// TIA Portal project "Semafoare_2026" (V15.1)

(* hardware
DEVICE "S71500/ET200MP station_1"  S7-1500 station
   slot 0: "Rail_0"  Rack  6ES7 590-1***0-0AA0
   slot 1: "PLC_1"  CPU 1513-1 PN  6ES7 513-1AL02-0AB0  V2.6
      slot 3: "CPU display_1"  6ES7591-1AA00-0AA0
DEVICE "HMI_1"  KTP900 Basic PN
   slot 0: "HMI_1"  KTP900 Basic PN  6AV2 123-2JB03-0AX0  15.1.0.0
   slot 1: "HMI_RT_1"  KTP900 Basic PN  6AV2 123-2JB03-0AX0  15.1.0.0
   slot 5: "HMI_1.IE_CP_1"  PROFINET Interface  15.0.1.0
      slot 1: "PROFINET Interface_1"  PROFINET Interface
         slot 1: "Port_1"  Port
*)

// ===== PLC "PLC_1"  CPU 1513-1 PN =====

VAR_GLOBAL   // PLC tag table "Default tag table"
   "Clock_Byte" AT %MB0 : Byte;
   "Clock_10Hz" AT %M0.0 : Bool;
   "Clock_5Hz" AT %M0.1 : Bool;
   "Clock_2.5Hz" AT %M0.2 : Bool;
   "Clock_2Hz" AT %M0.3 : Bool;
   "Clock_1.25Hz" AT %M0.4 : Bool;
   "Clock_1Hz" AT %M0.5 : Bool;
   "Clock_0.625Hz" AT %M0.6 : Bool;
   "Clock_0.5Hz" AT %M0.7 : Bool;
END_VAR

DATA_BLOCK "Semafor_masini_ciclu_DB"   // DB1
{ S7_Optimized_Access := 'TRUE' }
VERSION : 0.1
   VAR
      rosu_on : Bool;
      galben_on : Bool;
      galben_on_hmi : Bool;
      verde_on : Bool;
      time_elapsed_rosu : Time;
      time_elapsed_rosu_secunde : Time;
      time_elapsed_verde : Time;
      time_elapsed_verde_secunde : Time;
      time_elapsed_galben : Time;
      time_elapsed_galben_secunde : Time;
      "mod" : Int;
   END_VAR
BEGIN
END_DATA_BLOCK

DATA_BLOCK "Semafor_pietoni_DB"   // DB2
{ S7_Optimized_Access := 'TRUE' }
VERSION : 0.1
   VAR
      "mod" : Int;
      rosu_on : Bool;
      verde_on : Bool;
      time_elapsed_rosu : Time;
      time_elapsed_sec_rosu : Time;
      time_elapsed_verde : Time;
      time_elapsed_sec_verde : Time;
   END_VAR
BEGIN
END_DATA_BLOCK

DATA_BLOCK "Semafor_masini_ciclu_DB_1"   // DB3
{ S7_Optimized_Access := 'TRUE' }
VERSION : 0.1
// stored: InstanceOfName Semafor_masini_ciclu
"Semafor_masini_ciclu"
BEGIN
END_DATA_BLOCK

DATA_BLOCK "Semafor_pietoni_DB_1"   // DB4
{ S7_Optimized_Access := 'TRUE' }
VERSION : 0.1
// stored: InstanceOfName Semafor_pietoni
"Semafor_pietoni"
BEGIN
END_DATA_BLOCK

DATA_BLOCK "Semafor_pietoni_buton_DB"   // DB5
{ S7_Optimized_Access := 'TRUE' }
VERSION : 0.1
   VAR
      "mod" : Int;
      rosu_on : Bool;
      verde_on : Bool;
      buton : Bool;
      timer_buton_gata : Bool;
      intermitent_hmi : Bool;
      vizibil_hmi : Bool;
      time_elapsed_verde : Time;
      time_elapsed_sec_verde : Time;
      timp_intre : Time;
      timp_intre_sec : Time;
   END_VAR
BEGIN
END_DATA_BLOCK

DATA_BLOCK "Semafor_pietoni_buton_DB_1"   // DB6
{ S7_Optimized_Access := 'TRUE' }
VERSION : 0.1
// stored: InstanceOfName Semafor_pietoni_buton
"Semafor_pietoni_buton"
BEGIN
END_DATA_BLOCK

DATA_BLOCK "Semafor_masina_pietoni_DB"   // DB7
{ S7_Optimized_Access := 'TRUE' }
VERSION : 0.1
   VAR
      "mod" : Int;
      timer_buton_gata : Bool;
      buton : Bool;
      verde_on : Bool;
      rosu_on : Bool;
      galben_on : Bool;
      galben_on_hmi : Bool;
      pieton_verde_on : Bool;
      pieton_rosu_on : Bool;
      intermitent_hmi : Bool;
      vizibil_hmi : Bool;
      time_elapsed_galben : Time;
      time_elapsed_galben_sec : Time;
      time_elapsed_rosu : Time;
      time_elapsed_rosu_sec : Time;
      pieton_time_elapsed_verde : Time;
      pieton_time_elapsed_verde_sec : Time;
      time_intre : Time;
      time_buton : Time;
   END_VAR
BEGIN
END_DATA_BLOCK

DATA_BLOCK "Semafor_masina_buton_DB"   // DB8
{ S7_Optimized_Access := 'TRUE' }
VERSION : 0.1
   VAR
      verde_on : Bool;
      rosu_on : Bool;
      galben_on : Bool;
      galben_on_hmi : Bool;
      time_elapsed_galben : Time;
      time_elapsed_rosu : Time;
      time_elapsed_galben_sec : Time;
      tine_elapsed_rosu_sec : Time;
   END_VAR
BEGIN
END_DATA_BLOCK

DATA_BLOCK "Semafor_masina_buton_DB_1"   // DB9
{ S7_Optimized_Access := 'TRUE' }
VERSION : 0.1
// stored: InstanceOfName Semafor_masina_buton
"Semafor_masina_buton"
BEGIN
END_DATA_BLOCK

DATA_BLOCK "Semafor_masina_pietoni_DB_1"   // DB10
{ S7_Optimized_Access := 'TRUE' }
VERSION : 0.1
// stored: InstanceOfName Semafor_masina_pietoni
"Semafor_masina_pietoni"
BEGIN
END_DATA_BLOCK

DATA_BLOCK "Semafor_masina_buton_DB_2"   // DB11
{ S7_Optimized_Access := 'TRUE' }
VERSION : 0.1
// stored: InstanceOfName Semafor_masina_buton
"Semafor_masina_buton"
BEGIN
END_DATA_BLOCK

DATA_BLOCK "Semafor_pietoni_buton_DB_2"   // DB12
{ S7_Optimized_Access := 'TRUE' }
VERSION : 0.1
// stored: InstanceOfName Semafor_pietoni_buton
"Semafor_pietoni_buton"
BEGIN
END_DATA_BLOCK

DATA_BLOCK "Clock_custom_0.7Hz_DB"   // DB13
{ S7_Optimized_Access := 'TRUE' }
VERSION : 0.1
// stored: InstanceOfName Clock_custom_0.7Hz
"Clock_custom_0.7Hz"
BEGIN
END_DATA_BLOCK

DATA_BLOCK "test"   // DB14
{ S7_Optimized_Access := 'TRUE' }
VERSION : 0.1
   VAR
      activ : Bool;
      re : Bool;
      "counter" : Int;
   END_VAR
BEGIN
END_DATA_BLOCK

DATA_BLOCK "Buzzer_DB"   // DB15
{ S7_Optimized_Access := 'TRUE' }
VERSION : 0.1
   VAR
      permisiune_plecare : Bool;
      pornire_sunet : Bool;
   END_VAR
BEGIN
END_DATA_BLOCK

DATA_BLOCK "Buzzer_DB_1"   // DB16
{ S7_Optimized_Access := 'TRUE' }
VERSION : 0.1
// stored: InstanceOfName Buzzer
"Buzzer"
BEGIN
END_DATA_BLOCK

DATA_BLOCK "Buzzer_Pieton_buton_DB"   // DB17
{ S7_Optimized_Access := 'TRUE' }
VERSION : 0.1
   VAR
      permisiune_plecare : Bool;
      pornire_sunet : Bool;
   END_VAR
BEGIN
END_DATA_BLOCK

DATA_BLOCK "Buzzer_pieton_Masina_buton_DB"   // DB18
{ S7_Optimized_Access := 'TRUE' }
VERSION : 0.1
   VAR
      permisiune_plecare : Bool;
      pornire_sunet : Bool;
   END_VAR
BEGIN
END_DATA_BLOCK

DATA_BLOCK "Buzzer_DB_2"   // DB19
{ S7_Optimized_Access := 'TRUE' }
VERSION : 0.1
// stored: InstanceOfName Buzzer
"Buzzer"
BEGIN
END_DATA_BLOCK

DATA_BLOCK "Buzzer_DB_3"   // DB20
{ S7_Optimized_Access := 'TRUE' }
VERSION : 0.1
// stored: InstanceOfName Buzzer
"Buzzer"
BEGIN
END_DATA_BLOCK

DATA_BLOCK "Semafoare-2-masini_DB"   // DB21
{ S7_Optimized_Access := 'TRUE' }
VERSION : 0.1
   VAR
      "mod" : Int;
      te_rosu_1 : Time;
      te_rosu_sec_1 : Time;
      te_rosu_2 : Time;
      te_rosu_sec_2 : Time;
      te_galben_1 : Time;
      te_galben_sec_1 : Time;
      te_galben_2 : Time;
      te_galben_sec_2 : Time;
      te_verde_1 : Time;
      te_verde_sec_1 : Time;
      te_verde_2 : Time;
      te_verde_sec_2 : Time;
      verde_on_1 : Bool;
      verde_on_2 : Bool;
      galben_on_1 : Bool;
      galben_hmi_on_1 : Bool;
      galben_on_2 : Bool;
      galben_hmi_on_2 : Bool;
      rosu_on_1 : Bool;
      rosu_on_2 : Bool;
   END_VAR
BEGIN
END_DATA_BLOCK

DATA_BLOCK "Semafoare-2-masini_DB_1"   // DB22
{ S7_Optimized_Access := 'TRUE' }
VERSION : 0.1
// stored: InstanceOfName Semafoare-2-masini
"Semafoare-2-masini"
BEGIN
END_DATA_BLOCK

DATA_BLOCK "Semafor_masini_ciclu_DB_2"   // DB23
{ S7_Optimized_Access := 'TRUE' }
VERSION : 0.1
// stored: InstanceOfName Semafor_masini_ciclu
"Semafor_masini_ciclu"
BEGIN
END_DATA_BLOCK

DATA_BLOCK "Semafor_masini_ciclu_DB_3"   // DB24
{ S7_Optimized_Access := 'TRUE' }
VERSION : 0.1
// stored: InstanceOfName Semafor_masini_ciclu
"Semafor_masini_ciclu"
BEGIN
END_DATA_BLOCK

DATA_BLOCK "Semafor_masini_1_DB"   // DB25
{ S7_Optimized_Access := 'TRUE' }
VERSION : 0.1
// stored: InstanceOfName Semafor_masini_1
"Semafor_masini_1"
BEGIN
END_DATA_BLOCK

DATA_BLOCK "Semafor_masina_2_DB"   // DB26
{ S7_Optimized_Access := 'TRUE' }
VERSION : 0.1
// stored: InstanceOfName Semafor_masina_2
"Semafor_masina_2"
BEGIN
END_DATA_BLOCK

FUNCTION_BLOCK "Semafor_masini_ciclu"   // FB1, LAD
{ S7_Optimized_Access := 'TRUE' }
VERSION : 0.1
   VAR_INPUT
      mod_functinare : Int;
   END_VAR
   VAR_OUTPUT
      time_elapsed_verde : Time;
      time_elapsed_galben : Time;
      time_elapsed_rosu : Time;
   END_VAR
   VAR_IN_OUT
      verde_on : Bool;
      rosu_on : Bool;
      galben_on : Bool;
   END_VAR
   VAR
      timer_rosu : TON_TIME;
      timer_galben : TON_TIME;
      timer_verde : TON_TIME;
      galben_intermitent_on : Bool;
      re1 : Bool;
      re_aux : Bool;
      mod_normal : Bool;
      reseteaza_ciclul : Bool;
      porneste_verde : Bool;
      porneste_rosu : Bool;
      porneste_galben : Bool;
   END_VAR
   VAR_TEMP   // added for the SCL form of the ladder/FBD networks
      _w1 : Bool;
   END_VAR
BEGIN

REGION Network 1: semafor modul normal/mod oprire
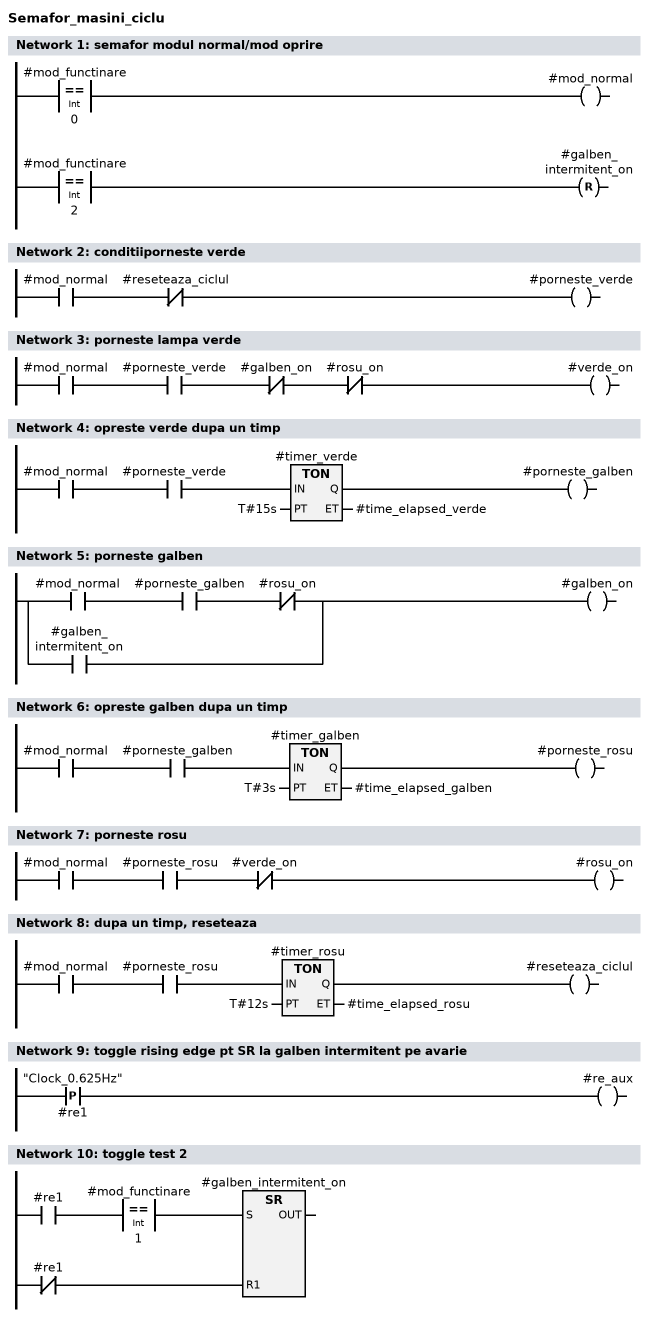
   RUNG wire#powerrail
      { S7_Templates := "SrcType := Int" } EQ_Contact(in1 := #mod_functinare, in2 := 0)
      Coil( #mod_normal )
   END_RUNG
   RUNG wire#powerrail
      { S7_Templates := "SrcType := Int" } EQ_Contact(in1 := #mod_functinare, in2 := 2)
      R_Coil( #galben_intermitent_on )
   END_RUNG
   // the same network as SCL:
   #mod_normal := #mod_functinare = 0;
   IF #mod_functinare = 2 THEN #galben_intermitent_on := FALSE; END_IF;
END_REGION

REGION Network 2: conditiiporneste verde
   RUNG wire#powerrail
      Contact( #mod_normal )
      I_Contact( #reseteaza_ciclul )
      Coil( #porneste_verde )
   END_RUNG
   // the same network as SCL:
   #porneste_verde := #mod_normal AND NOT #reseteaza_ciclul;
END_REGION

REGION Network 3: porneste lampa verde
   RUNG wire#powerrail
      Contact( #mod_normal )
      Contact( #porneste_verde )
      I_Contact( #galben_on )
      I_Contact( #rosu_on )
      Coil( #verde_on )
   END_RUNG
   // the same network as SCL:
   #verde_on := #mod_normal AND #porneste_verde AND NOT #galben_on AND NOT #rosu_on;
END_REGION

REGION Network 4: opreste verde dupa un timp
   #timer_verde(IN := #mod_normal AND #porneste_verde, PT := T#15s, ET => #time_elapsed_verde);   // TON
   #porneste_galben := #timer_verde.Q;
END_REGION

REGION Network 5: porneste galben
   RUNG wire#powerrail
      Contact( #mod_normal )
      Contact( #porneste_galben )
      I_Contact( #rosu_on )
      wire#w1
      Coil( #galben_on )
   END_RUNG
   RUNG wire#powerrail
      Contact( #galben_intermitent_on )
   END_RUNG wire#w1
   // the same network as SCL:
   #galben_on := (#mod_normal AND #porneste_galben AND NOT #rosu_on) OR #galben_intermitent_on;
END_REGION

REGION Network 6: opreste galben dupa un timp
   #timer_galben(IN := #mod_normal AND #porneste_galben, PT := T#3s, ET => #time_elapsed_galben);   // TON
   #porneste_rosu := #timer_galben.Q;
END_REGION

REGION Network 7: porneste rosu
   RUNG wire#powerrail
      Contact( #mod_normal )
      Contact( #porneste_rosu )
      I_Contact( #verde_on )
      Coil( #rosu_on )
   END_RUNG
   // the same network as SCL:
   #rosu_on := #mod_normal AND #porneste_rosu AND NOT #verde_on;
END_REGION

REGION Network 8: dupa un timp, reseteaza
   #timer_rosu(IN := #mod_normal AND #porneste_rosu, PT := T#12s, ET => #time_elapsed_rosu);   // TON
   #reseteaza_ciclul := #timer_rosu.Q;
END_REGION

REGION Network 9: toggle rising edge pt SR la galben intermitent pe avarie
   RUNG wire#powerrail
      P_Contact(operand := "Clock_0.625Hz", bit := #re1)
      Coil( #re_aux )
   END_RUNG
   // the same network as SCL:
   #_w1 := "Clock_0.625Hz" AND NOT #re1;   // rising edge of "Clock_0.625Hz"
   #re1 := "Clock_0.625Hz";
   #re_aux := #_w1;
END_REGION

REGION Network 10: toggle test 2
   RUNG wire#powerrail
      Contact( #re1 )
      { S7_Templates := "SrcType := Int" } EQ_Contact(in1 := #mod_functinare, in2 := 1)
      S_SR(operand := #galben_intermitent_on, r1 := wire#w1)
   END_RUNG
   RUNG wire#powerrail
      I_Contact( #re1 )
   END_RUNG wire#w1
   // the same network as SCL:
   IF #re1 AND (#mod_functinare = 1) THEN
       #galben_intermitent_on := TRUE;   // SR flip-flop
   END_IF;
   IF NOT #re1 THEN #galben_intermitent_on := FALSE; END_IF;
END_REGION
END_FUNCTION_BLOCK

FUNCTION_BLOCK "Semafor_pietoni"   // FB2, LAD
{ S7_Optimized_Access := 'TRUE' }
VERSION : 0.1
   VAR_INPUT
      "mod" : Int;
   END_VAR
   VAR_OUTPUT
      verde_on : Bool;
      rosu_on : Bool;
      time_elapsed_verde : Time;
      time_elapsed_rosu : Time;
   END_VAR
   VAR
      timer_verde : TON_TIME;
      timer_rosu : TON_TIME;
      reseteaza_ciclul : Bool;
      porneste_verde : Bool;
      porneste_rosu : Bool;
   END_VAR
BEGIN

REGION Network 1: conditii sa porneasca verde
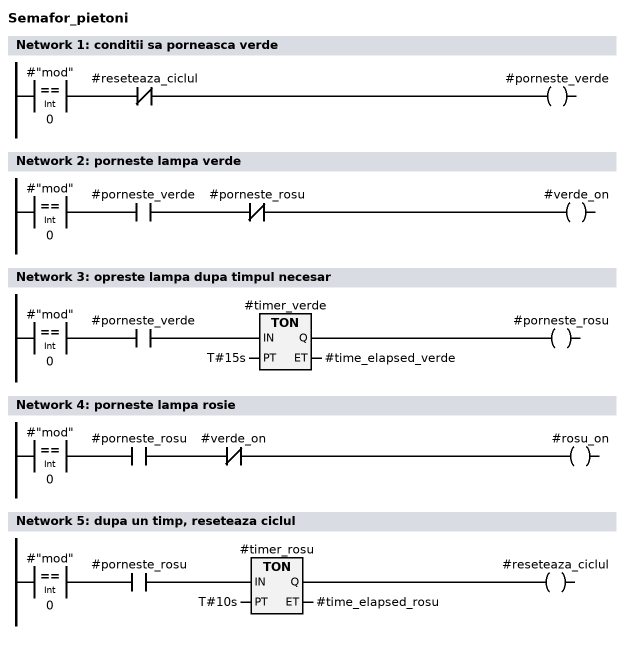
   RUNG wire#powerrail
      { S7_Templates := "SrcType := Int" } EQ_Contact(in1 := #"mod", in2 := 0)
      I_Contact( #reseteaza_ciclul )
      Coil( #porneste_verde )
   END_RUNG
   // the same network as SCL:
   #porneste_verde := (#"mod" = 0) AND NOT #reseteaza_ciclul;
END_REGION

REGION Network 2: porneste lampa verde
   RUNG wire#powerrail
      { S7_Templates := "SrcType := Int" } EQ_Contact(in1 := #"mod", in2 := 0)
      Contact( #porneste_verde )
      I_Contact( #porneste_rosu )
      Coil( #verde_on )
   END_RUNG
   // the same network as SCL:
   #verde_on := (#"mod" = 0) AND #porneste_verde AND NOT #porneste_rosu;
END_REGION

REGION Network 3: opreste lampa dupa timpul necesar
   #timer_verde(IN := (#"mod" = 0) AND #porneste_verde, PT := T#15s, ET => #time_elapsed_verde);   // TON
   #porneste_rosu := #timer_verde.Q;
END_REGION

REGION Network 4: porneste lampa rosie
   RUNG wire#powerrail
      { S7_Templates := "SrcType := Int" } EQ_Contact(in1 := #"mod", in2 := 0)
      Contact( #porneste_rosu )
      I_Contact( #verde_on )
      Coil( #rosu_on )
   END_RUNG
   // the same network as SCL:
   #rosu_on := (#"mod" = 0) AND #porneste_rosu AND NOT #verde_on;
END_REGION

REGION Network 5: dupa un timp, reseteaza ciclul
   #timer_rosu(IN := (#"mod" = 0) AND #porneste_rosu, PT := T#10s, ET => #time_elapsed_rosu);   // TON
   #reseteaza_ciclul := #timer_rosu.Q;
END_REGION
END_FUNCTION_BLOCK

FUNCTION_BLOCK "Semafor_pietoni_buton"   // FB3, LAD
{ S7_Optimized_Access := 'TRUE' }
VERSION : 0.1
   VAR_INPUT
      "mod" : Int;
      rosu_masina_on : Bool;
   END_VAR
   VAR_OUTPUT
      verde_on : Bool;
      rosu_on : Bool;
      time_elapsed_verde : Time;
      time_intre : Time;
      time_buton : Time;
      intermitent_hmi : Bool;
      vizibil_hmi : Bool;
   END_VAR
   VAR_IN_OUT
      buton : Bool;
      timer_buton_gata : Bool;
   END_VAR
   VAR
      timer_verde : TON_TIME;
      timer_intre : TON_TIME;
      timer_buton : TON_TIME;
      porneste_verde : Bool;
      porneste_rosu : Bool;
      temp : Bool;
      re_aux : Bool;
      re : Bool;
      gata_verde : Bool;
   END_VAR
   VAR_TEMP   // added for the SCL form of the ladder/FBD networks
      _w1 : Bool;
   END_VAR
BEGIN

REGION Network 1: conditia sa ramana rosu pornit
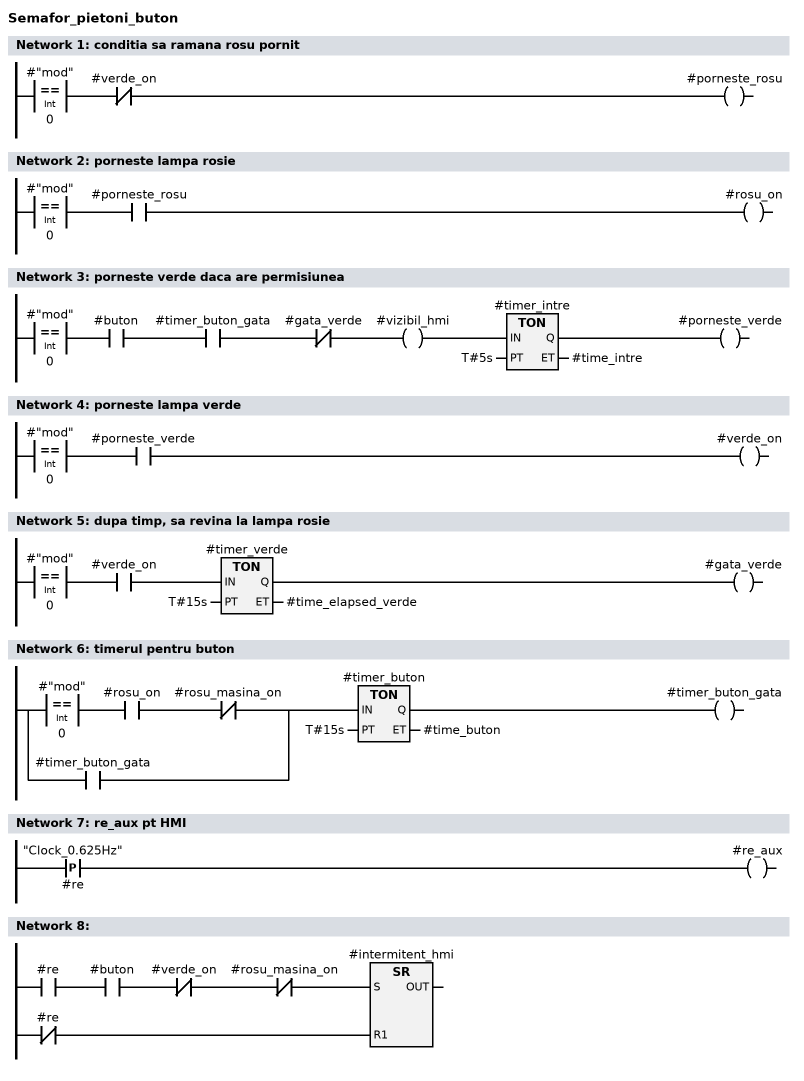
   RUNG wire#powerrail
      { S7_Templates := "SrcType := Int" } EQ_Contact(in1 := #"mod", in2 := 0)
      I_Contact( #verde_on )
      Coil( #porneste_rosu )
   END_RUNG
   // the same network as SCL:
   #porneste_rosu := (#"mod" = 0) AND NOT #verde_on;
END_REGION

REGION Network 2: porneste lampa rosie
   RUNG wire#powerrail
      { S7_Templates := "SrcType := Int" } EQ_Contact(in1 := #"mod", in2 := 0)
      Contact( #porneste_rosu )
      Coil( #rosu_on )
   END_RUNG
   // the same network as SCL:
   #rosu_on := (#"mod" = 0) AND #porneste_rosu;
END_REGION

REGION Network 3: porneste verde daca are permisiunea
   #vizibil_hmi := (#"mod" = 0) AND #buton AND #timer_buton_gata AND NOT #gata_verde;
   #timer_intre(IN := #vizibil_hmi, PT := T#5s, ET => #time_intre);   // TON
   #porneste_verde := #timer_intre.Q;
END_REGION

REGION Network 4: porneste lampa verde
   RUNG wire#powerrail
      { S7_Templates := "SrcType := Int" } EQ_Contact(in1 := #"mod", in2 := 0)
      Contact( #porneste_verde )
      Coil( #verde_on )
   END_RUNG
   // the same network as SCL:
   #verde_on := (#"mod" = 0) AND #porneste_verde;
END_REGION

REGION Network 5: dupa timp, sa revina la lampa rosie
   #timer_verde(IN := (#"mod" = 0) AND #verde_on, PT := T#15s, ET => #time_elapsed_verde);   // TON
   #gata_verde := #timer_verde.Q;
END_REGION

REGION Network 6: timerul pentru buton
   #timer_buton(IN := ((#"mod" = 0) AND #rosu_on AND NOT #rosu_masina_on) OR #timer_buton_gata,   // TON
                PT := T#15s,
                ET => #time_buton);
   #timer_buton_gata := #timer_buton.Q;
END_REGION

REGION Network 7: re_aux pt HMI
   RUNG wire#powerrail
      P_Contact(operand := "Clock_0.625Hz", bit := #re)
      Coil( #re_aux )
   END_RUNG
   // the same network as SCL:
   #_w1 := "Clock_0.625Hz" AND NOT #re;   // rising edge of "Clock_0.625Hz"
   #re := "Clock_0.625Hz";
   #re_aux := #_w1;
END_REGION

REGION Network 8
   RUNG wire#powerrail
      Contact( #re )
      Contact( #buton )
      I_Contact( #verde_on )
      I_Contact( #rosu_masina_on )
      S_SR(operand := #intermitent_hmi, r1 := wire#w1)
   END_RUNG
   RUNG wire#powerrail
      I_Contact( #re )
   END_RUNG wire#w1
   // the same network as SCL:
   IF #re AND #buton AND NOT #verde_on AND NOT #rosu_masina_on THEN
       #intermitent_hmi := TRUE;   // SR flip-flop
   END_IF;
   IF NOT #re THEN #intermitent_hmi := FALSE; END_IF;
END_REGION
END_FUNCTION_BLOCK

FUNCTION_BLOCK "Semafor_masina_pietoni"   // FB4, LAD
{ S7_Optimized_Access := 'TRUE' }
VERSION : 0.1
   VAR_INPUT
      "mod" : Int;
   END_VAR
   VAR_OUTPUT
      pornire_sunet_buzzer : Bool;
      time_elapsed_galben : Time;
      time_elapsed_rosu : Time;
      pieton_time_elapsed_verde : Time;
      time_intre : Time;
      time_buton : Time;
      intermitent_hmi : Bool;
      vizibil_hmi : Bool;
   END_VAR
   VAR_IN_OUT
      permisiune_plecare_buzzer : Bool;
      timer_buton_gata : Bool;
      buton : Bool;
      verde_on : Bool;
      rosu_on : Bool;
      galben_on : Bool;
      pieton_verde_on : Bool;
      pieton_rosu_on : Bool;
   END_VAR
BEGIN

REGION Network 1: semafor masina
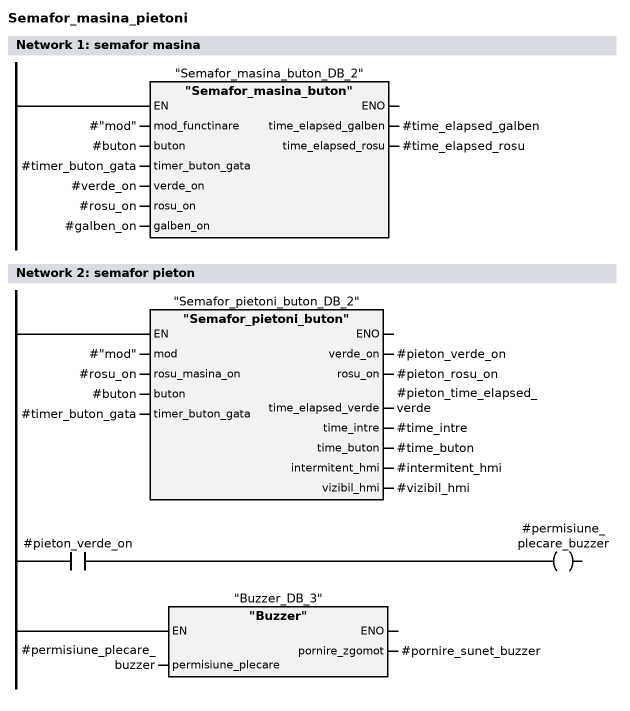
   RUNG wire#powerrail
      "Semafor_masina_buton_DB_2"(mod_functinare := #"mod", buton := #buton, timer_buton_gata := #timer_buton_gata, verde_on := #verde_on, rosu_on := #rosu_on, galben_on := #galben_on, time_elapsed_galben => #time_elapsed_galben, time_elapsed_rosu => #time_elapsed_rosu)
   END_RUNG
   // the same network as SCL:
   "Semafor_masina_buton_DB_2"(mod_functinare := #"mod",   // "Semafor_masina_buton"
                           buton := #buton,
                           timer_buton_gata := #timer_buton_gata,
                           verde_on := #verde_on,
                           rosu_on := #rosu_on,
                           galben_on := #galben_on,
                           time_elapsed_galben => #time_elapsed_galben,
                           time_elapsed_rosu => #time_elapsed_rosu);
END_REGION

REGION Network 2: semafor pieton
   RUNG wire#powerrail
      "Semafor_pietoni_buton_DB_2"("mod" := #"mod", rosu_masina_on := #rosu_on, buton := #buton, timer_buton_gata := #timer_buton_gata, verde_on => #pieton_verde_on, rosu_on => #pieton_rosu_on, time_elapsed_verde => #pieton_time_elapsed_verde, time_intre => #time_intre, time_buton => #time_buton, intermitent_hmi => #intermitent_hmi, vizibil_hmi => #vizibil_hmi)
   END_RUNG
   RUNG wire#powerrail
      Contact( #pieton_verde_on )
      Coil( #permisiune_plecare_buzzer )
   END_RUNG
   RUNG wire#powerrail
      "Buzzer_DB_3"(permisiune_plecare := #permisiune_plecare_buzzer, pornire_zgomot => #pornire_sunet_buzzer)
   END_RUNG
   // the same network as SCL:
   "Semafor_pietoni_buton_DB_2"("mod" := #"mod",   // "Semafor_pietoni_buton"
                           rosu_masina_on := #rosu_on,
                           buton := #buton,
                           timer_buton_gata := #timer_buton_gata,
                           verde_on => #pieton_verde_on,
                           rosu_on => #pieton_rosu_on,
                           time_elapsed_verde => #pieton_time_elapsed_verde,
                           time_intre => #time_intre,
                           time_buton => #time_buton,
                           intermitent_hmi => #intermitent_hmi,
                           vizibil_hmi => #vizibil_hmi);
   #permisiune_plecare_buzzer := #pieton_verde_on;
   "Buzzer_DB_3"(permisiune_plecare := #permisiune_plecare_buzzer, pornire_zgomot => #pornire_sunet_buzzer);   // "Buzzer"
END_REGION
END_FUNCTION_BLOCK

FUNCTION_BLOCK "Semafor_masina_buton"   // FB5, LAD
{ S7_Optimized_Access := 'TRUE' }
VERSION : 0.1
   VAR_INPUT
      mod_functinare : Int;
   END_VAR
   VAR_OUTPUT
      time_elapsed_galben : Time;
      time_elapsed_rosu : Time;
   END_VAR
   VAR_IN_OUT
      buton : Bool;
      timer_buton_gata : Bool;
      verde_on : Bool;
      rosu_on : Bool;
      galben_on : Bool;
   END_VAR
   VAR
      timer_rosu : TON_TIME;
      timer_galben : TON_TIME;
      galben_intermitent_on : Bool;
      re1 : Bool;
      re_aux : Bool;
      porneste_verde : Bool;
      porneste_rosu : Bool;
      porneste_galben : Bool;
   END_VAR
   VAR_TEMP   // added for the SCL form of the ladder/FBD networks
      _w1 : Bool;
   END_VAR
BEGIN

REGION Network 1: conditia sa ramana verde pornit
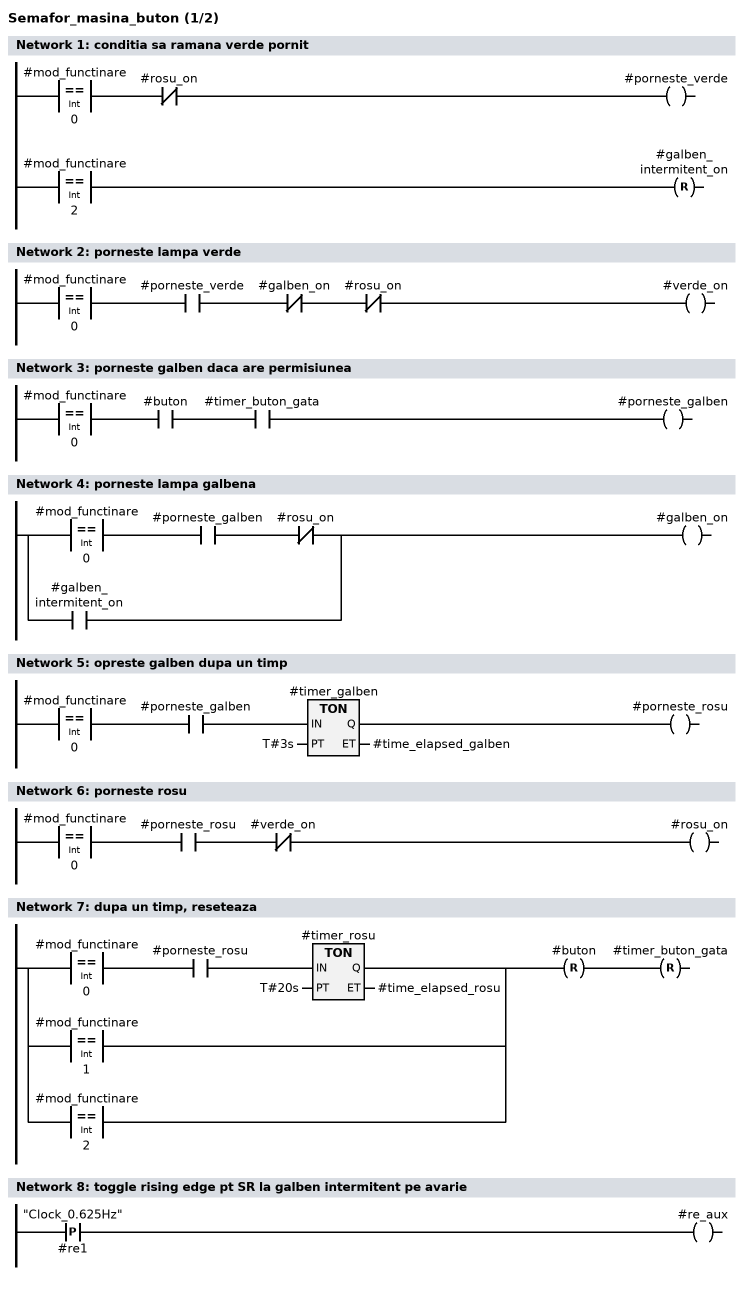
   RUNG wire#powerrail
      { S7_Templates := "SrcType := Int" } EQ_Contact(in1 := #mod_functinare, in2 := 0)
      I_Contact( #rosu_on )
      Coil( #porneste_verde )
   END_RUNG
   RUNG wire#powerrail
      { S7_Templates := "SrcType := Int" } EQ_Contact(in1 := #mod_functinare, in2 := 2)
      R_Coil( #galben_intermitent_on )
   END_RUNG
   // the same network as SCL:
   #porneste_verde := (#mod_functinare = 0) AND NOT #rosu_on;
   IF #mod_functinare = 2 THEN #galben_intermitent_on := FALSE; END_IF;
END_REGION

REGION Network 2: porneste lampa verde
   RUNG wire#powerrail
      { S7_Templates := "SrcType := Int" } EQ_Contact(in1 := #mod_functinare, in2 := 0)
      Contact( #porneste_verde )
      I_Contact( #galben_on )
      I_Contact( #rosu_on )
      Coil( #verde_on )
   END_RUNG
   // the same network as SCL:
   #verde_on := (#mod_functinare = 0) AND #porneste_verde AND NOT #galben_on AND NOT #rosu_on;
END_REGION

REGION Network 3: porneste galben daca are permisiunea
   RUNG wire#powerrail
      { S7_Templates := "SrcType := Int" } EQ_Contact(in1 := #mod_functinare, in2 := 0)
      Contact( #buton )
      Contact( #timer_buton_gata )
      Coil( #porneste_galben )
   END_RUNG
   // the same network as SCL:
   #porneste_galben := (#mod_functinare = 0) AND #buton AND #timer_buton_gata;
END_REGION

REGION Network 4: porneste lampa galbena
   RUNG wire#powerrail
      { S7_Templates := "SrcType := Int" } EQ_Contact(in1 := #mod_functinare, in2 := 0)
      Contact( #porneste_galben )
      I_Contact( #rosu_on )
      wire#w1
      Coil( #galben_on )
   END_RUNG
   RUNG wire#powerrail
      Contact( #galben_intermitent_on )
   END_RUNG wire#w1
   // the same network as SCL:
   #galben_on := ((#mod_functinare = 0) AND #porneste_galben AND NOT #rosu_on) OR #galben_intermitent_on;
END_REGION

REGION Network 5: opreste galben dupa un timp
   #timer_galben(IN := (#mod_functinare = 0) AND #porneste_galben, PT := T#3s, ET => #time_elapsed_galben);   // TON
   #porneste_rosu := #timer_galben.Q;
END_REGION

REGION Network 6: porneste rosu
   RUNG wire#powerrail
      { S7_Templates := "SrcType := Int" } EQ_Contact(in1 := #mod_functinare, in2 := 0)
      Contact( #porneste_rosu )
      I_Contact( #verde_on )
      Coil( #rosu_on )
   END_RUNG
   // the same network as SCL:
   #rosu_on := (#mod_functinare = 0) AND #porneste_rosu AND NOT #verde_on;
END_REGION

REGION Network 7: dupa un timp, reseteaza
   #timer_rosu(IN := (#mod_functinare = 0) AND #porneste_rosu, PT := T#20s, ET => #time_elapsed_rosu);   // TON
   IF #timer_rosu.Q OR (#mod_functinare = 1) OR (#mod_functinare = 2) THEN
       #buton := FALSE;
       #timer_buton_gata := FALSE;
   END_IF;
END_REGION

REGION Network 8: toggle rising edge pt SR la galben intermitent pe avarie
   RUNG wire#powerrail
      P_Contact(operand := "Clock_0.625Hz", bit := #re1)
      Coil( #re_aux )
   END_RUNG
   // the same network as SCL:
   #_w1 := "Clock_0.625Hz" AND NOT #re1;   // rising edge of "Clock_0.625Hz"
   #re1 := "Clock_0.625Hz";
   #re_aux := #_w1;
END_REGION

REGION Network 9: toggle test 2
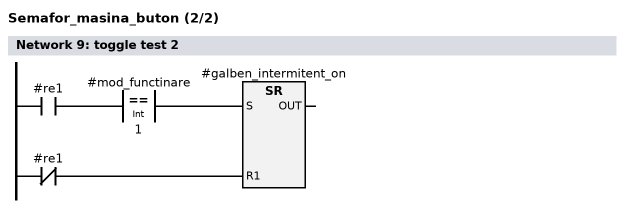
   RUNG wire#powerrail
      Contact( #re1 )
      { S7_Templates := "SrcType := Int" } EQ_Contact(in1 := #mod_functinare, in2 := 1)
      S_SR(operand := #galben_intermitent_on, r1 := wire#w1)
   END_RUNG
   RUNG wire#powerrail
      I_Contact( #re1 )
   END_RUNG wire#w1
   // the same network as SCL:
   IF #re1 AND (#mod_functinare = 1) THEN
       #galben_intermitent_on := TRUE;   // SR flip-flop
   END_IF;
   IF NOT #re1 THEN #galben_intermitent_on := FALSE; END_IF;
END_REGION
END_FUNCTION_BLOCK

FUNCTION_BLOCK "Clock_custom_0.7Hz"   // FB6, LAD
{ S7_Optimized_Access := 'TRUE' }
VERSION : 0.1
   VAR_OUTPUT
      activ : Bool;
   END_VAR
   VAR
      re : Bool;
      "counter" : Int;
   END_VAR
   VAR_TEMP   // added for the SCL form of the ladder/FBD networks
      _w1 : Bool;
   END_VAR
BEGIN

REGION Network 1
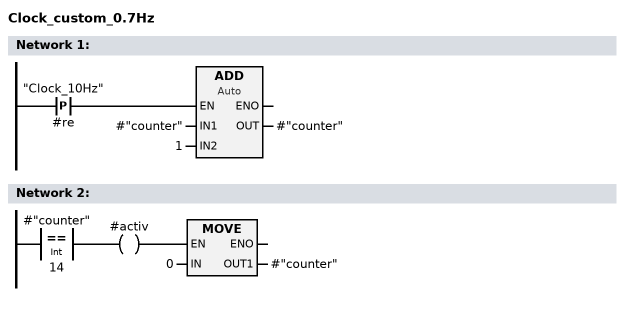
   RUNG wire#powerrail
      P_Contact(operand := "Clock_10Hz", bit := #re)
      Add(in1 := #"counter", in2 := 1, out => #"counter")
   END_RUNG
   // the same network as SCL:
   #_w1 := "Clock_10Hz" AND NOT #re;   // rising edge of "Clock_10Hz"
   #re := "Clock_10Hz";
   IF #_w1 THEN #"counter" := #"counter" + 1; END_IF;
END_REGION

REGION Network 2
   RUNG wire#powerrail
      { S7_Templates := "SrcType := Int" } EQ_Contact(in1 := #"counter", in2 := 14)
      Coil( #activ )
      Move(in := 0, out1 => #"counter")
   END_RUNG
   // the same network as SCL:
   #activ := #"counter" = 14;
   IF #activ THEN #"counter" := 0; END_IF;
END_REGION
END_FUNCTION_BLOCK

FUNCTION_BLOCK "Buzzer"   // FB7, LAD
{ S7_Optimized_Access := 'TRUE' }
VERSION : 0.1
   VAR_INPUT
      permisiune_plecare : Bool;
   END_VAR
   VAR_OUTPUT
      pornire_zgomot : Bool;
   END_VAR
   VAR
      re_aux : Bool;
      re : Bool;
   END_VAR
   VAR_TEMP   // added for the SCL form of the ladder/FBD networks
      _w1 : Bool;
   END_VAR
BEGIN

REGION Network 1: Auxiliara pentru SR
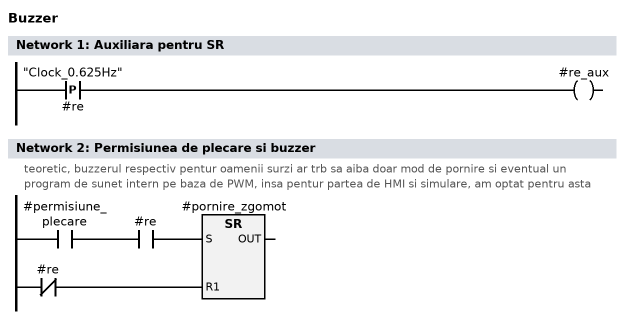
   RUNG wire#powerrail
      P_Contact(operand := "Clock_0.625Hz", bit := #re)
      Coil( #re_aux )
   END_RUNG
   // the same network as SCL:
   #_w1 := "Clock_0.625Hz" AND NOT #re;   // rising edge of "Clock_0.625Hz"
   #re := "Clock_0.625Hz";
   #re_aux := #_w1;
END_REGION

REGION Network 2: Permisiunea de plecare si buzzer
   // teoretic, buzzerul respectiv pentur oamenii surzi ar trb sa aiba doar mod de pornire si eventual un program de sunet intern pe baza de PWM, insa pentur partea de HMI si simulare, am optat pentru asta
   RUNG wire#powerrail
      Contact( #permisiune_plecare )
      Contact( #re )
      S_SR(operand := #pornire_zgomot, r1 := wire#w1)
   END_RUNG
   RUNG wire#powerrail
      I_Contact( #re )
   END_RUNG wire#w1
   // the same network as SCL:
   IF #permisiune_plecare AND #re THEN
       #pornire_zgomot := TRUE;   // SR flip-flop
   END_IF;
   IF NOT #re THEN #pornire_zgomot := FALSE; END_IF;
END_REGION
END_FUNCTION_BLOCK

FUNCTION_BLOCK "Semafoare-2-masini"   // FB8, LAD
{ S7_Optimized_Access := 'TRUE' }
VERSION : 0.1
   VAR_INPUT
      "mod" : Int;
   END_VAR
   VAR_OUTPUT
      te_rosu_1 : Time;
      te_rosu_2 : Time;
      te_galben_1 : Time;
      te_galben_2 : Time;
      te_verde_1 : Time;
      te_verde_2 : Time;
   END_VAR
   VAR_IN_OUT
      verde_on_1 : Bool;
      verde_on_2 : Bool;
      galben_on_1 : Bool;
      galben_on_2 : Bool;
      rosu_on_1 : Bool;
      rosu_on_2 : Bool;
   END_VAR
BEGIN

REGION Network 1: semafor masini 1
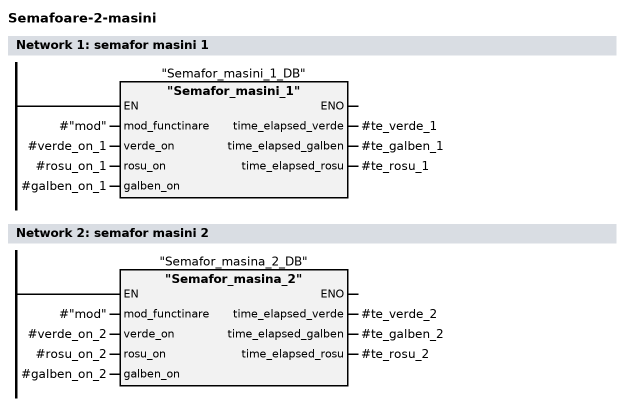
   RUNG wire#powerrail
      "Semafor_masini_1_DB"(mod_functinare := #"mod", verde_on := #verde_on_1, rosu_on := #rosu_on_1, galben_on := #galben_on_1, time_elapsed_verde => #te_verde_1, time_elapsed_galben => #te_galben_1, time_elapsed_rosu => #te_rosu_1)
   END_RUNG
   // the same network as SCL:
   "Semafor_masini_1_DB"(mod_functinare := #"mod",   // "Semafor_masini_1"
                         verde_on := #verde_on_1,
                         rosu_on := #rosu_on_1,
                         galben_on := #galben_on_1,
                         time_elapsed_verde => #te_verde_1,
                         time_elapsed_galben => #te_galben_1,
                         time_elapsed_rosu => #te_rosu_1);
END_REGION

REGION Network 2: semafor masini 2
   RUNG wire#powerrail
      "Semafor_masina_2_DB"(mod_functinare := #"mod", verde_on := #verde_on_2, rosu_on := #rosu_on_2, galben_on := #galben_on_2, time_elapsed_verde => #te_verde_2, time_elapsed_galben => #te_galben_2, time_elapsed_rosu => #te_rosu_2)
   END_RUNG
   // the same network as SCL:
   "Semafor_masina_2_DB"(mod_functinare := #"mod",   // "Semafor_masina_2"
                         verde_on := #verde_on_2,
                         rosu_on := #rosu_on_2,
                         galben_on := #galben_on_2,
                         time_elapsed_verde => #te_verde_2,
                         time_elapsed_galben => #te_galben_2,
                         time_elapsed_rosu => #te_rosu_2);
END_REGION
END_FUNCTION_BLOCK

FUNCTION_BLOCK "Semafor_masini_1"   // FB9, LAD
{ S7_Optimized_Access := 'TRUE' }
VERSION : 0.1
   VAR_INPUT
      mod_functinare : Int;
   END_VAR
   VAR_OUTPUT
      time_elapsed_verde : Time;
      time_elapsed_galben : Time;
      time_elapsed_rosu : Time;
   END_VAR
   VAR_IN_OUT
      verde_on : Bool;
      rosu_on : Bool;
      galben_on : Bool;
   END_VAR
   VAR
      timer_rosu : TON_TIME;
      timer_galben : TON_TIME;
      timer_verde : TON_TIME;
      galben_intermitent_on : Bool;
      re1 : Bool;
      re_aux : Bool;
      mod_normal : Bool;
      reseteaza_ciclul : Bool;
      porneste_verde : Bool;
      porneste_rosu : Bool;
      porneste_galben : Bool;
   END_VAR
   VAR_TEMP   // added for the SCL form of the ladder/FBD networks
      _w1 : Bool;
   END_VAR
BEGIN

REGION Network 1: semafor modul normal/mod oprire
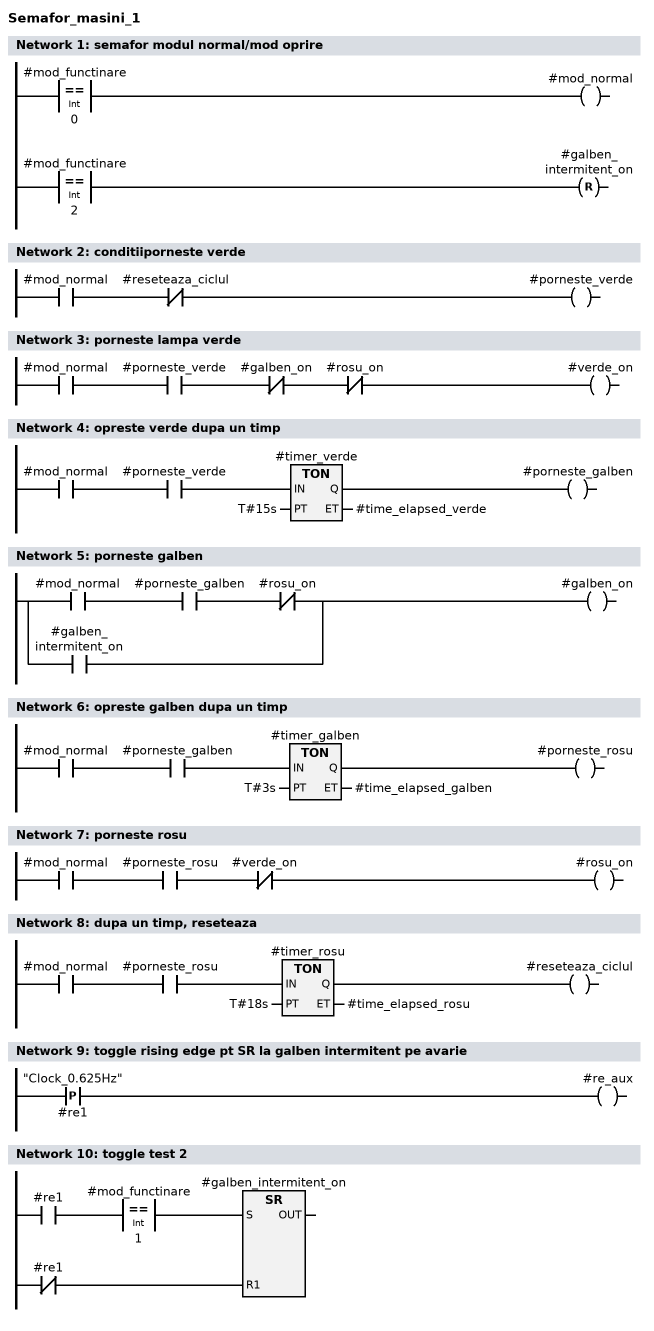
   RUNG wire#powerrail
      { S7_Templates := "SrcType := Int" } EQ_Contact(in1 := #mod_functinare, in2 := 0)
      Coil( #mod_normal )
   END_RUNG
   RUNG wire#powerrail
      { S7_Templates := "SrcType := Int" } EQ_Contact(in1 := #mod_functinare, in2 := 2)
      R_Coil( #galben_intermitent_on )
   END_RUNG
   // the same network as SCL:
   #mod_normal := #mod_functinare = 0;
   IF #mod_functinare = 2 THEN #galben_intermitent_on := FALSE; END_IF;
END_REGION

REGION Network 2: conditiiporneste verde
   RUNG wire#powerrail
      Contact( #mod_normal )
      I_Contact( #reseteaza_ciclul )
      Coil( #porneste_verde )
   END_RUNG
   // the same network as SCL:
   #porneste_verde := #mod_normal AND NOT #reseteaza_ciclul;
END_REGION

REGION Network 3: porneste lampa verde
   RUNG wire#powerrail
      Contact( #mod_normal )
      Contact( #porneste_verde )
      I_Contact( #galben_on )
      I_Contact( #rosu_on )
      Coil( #verde_on )
   END_RUNG
   // the same network as SCL:
   #verde_on := #mod_normal AND #porneste_verde AND NOT #galben_on AND NOT #rosu_on;
END_REGION

REGION Network 4: opreste verde dupa un timp
   #timer_verde(IN := #mod_normal AND #porneste_verde, PT := T#15s, ET => #time_elapsed_verde);   // TON
   #porneste_galben := #timer_verde.Q;
END_REGION

REGION Network 5: porneste galben
   RUNG wire#powerrail
      Contact( #mod_normal )
      Contact( #porneste_galben )
      I_Contact( #rosu_on )
      wire#w1
      Coil( #galben_on )
   END_RUNG
   RUNG wire#powerrail
      Contact( #galben_intermitent_on )
   END_RUNG wire#w1
   // the same network as SCL:
   #galben_on := (#mod_normal AND #porneste_galben AND NOT #rosu_on) OR #galben_intermitent_on;
END_REGION

REGION Network 6: opreste galben dupa un timp
   #timer_galben(IN := #mod_normal AND #porneste_galben, PT := T#3s, ET => #time_elapsed_galben);   // TON
   #porneste_rosu := #timer_galben.Q;
END_REGION

REGION Network 7: porneste rosu
   RUNG wire#powerrail
      Contact( #mod_normal )
      Contact( #porneste_rosu )
      I_Contact( #verde_on )
      Coil( #rosu_on )
   END_RUNG
   // the same network as SCL:
   #rosu_on := #mod_normal AND #porneste_rosu AND NOT #verde_on;
END_REGION

REGION Network 8: dupa un timp, reseteaza
   #timer_rosu(IN := #mod_normal AND #porneste_rosu, PT := T#18s, ET => #time_elapsed_rosu);   // TON
   #reseteaza_ciclul := #timer_rosu.Q;
END_REGION

REGION Network 9: toggle rising edge pt SR la galben intermitent pe avarie
   RUNG wire#powerrail
      P_Contact(operand := "Clock_0.625Hz", bit := #re1)
      Coil( #re_aux )
   END_RUNG
   // the same network as SCL:
   #_w1 := "Clock_0.625Hz" AND NOT #re1;   // rising edge of "Clock_0.625Hz"
   #re1 := "Clock_0.625Hz";
   #re_aux := #_w1;
END_REGION

REGION Network 10: toggle test 2
   RUNG wire#powerrail
      Contact( #re1 )
      { S7_Templates := "SrcType := Int" } EQ_Contact(in1 := #mod_functinare, in2 := 1)
      S_SR(operand := #galben_intermitent_on, r1 := wire#w1)
   END_RUNG
   RUNG wire#powerrail
      I_Contact( #re1 )
   END_RUNG wire#w1
   // the same network as SCL:
   IF #re1 AND (#mod_functinare = 1) THEN
       #galben_intermitent_on := TRUE;   // SR flip-flop
   END_IF;
   IF NOT #re1 THEN #galben_intermitent_on := FALSE; END_IF;
END_REGION
END_FUNCTION_BLOCK

FUNCTION_BLOCK "Semafor_masina_2"   // FB10, LAD
{ S7_Optimized_Access := 'TRUE' }
VERSION : 0.1
   VAR_INPUT
      mod_functinare : Int;
   END_VAR
   VAR_OUTPUT
      time_elapsed_verde : Time;
      time_elapsed_galben : Time;
      time_elapsed_rosu : Time;
   END_VAR
   VAR_IN_OUT
      verde_on : Bool;
      rosu_on : Bool;
      galben_on : Bool;
   END_VAR
   VAR
      timer_rosu : TON_TIME;
      timer_galben : TON_TIME;
      timer_verde : TON_TIME;
      galben_intermitent_on : Bool;
      re1 : Bool;
      re_aux : Bool;
      mod_normal : Bool;
      reseteaza_ciclul : Bool;
      porneste_verde : Bool;
      porneste_rosu : Bool;
      porneste_galben : Bool;
   END_VAR
   VAR_TEMP   // added for the SCL form of the ladder/FBD networks
      _w1 : Bool;
   END_VAR
BEGIN

REGION Network 1: semafor modul normal/mod oprire
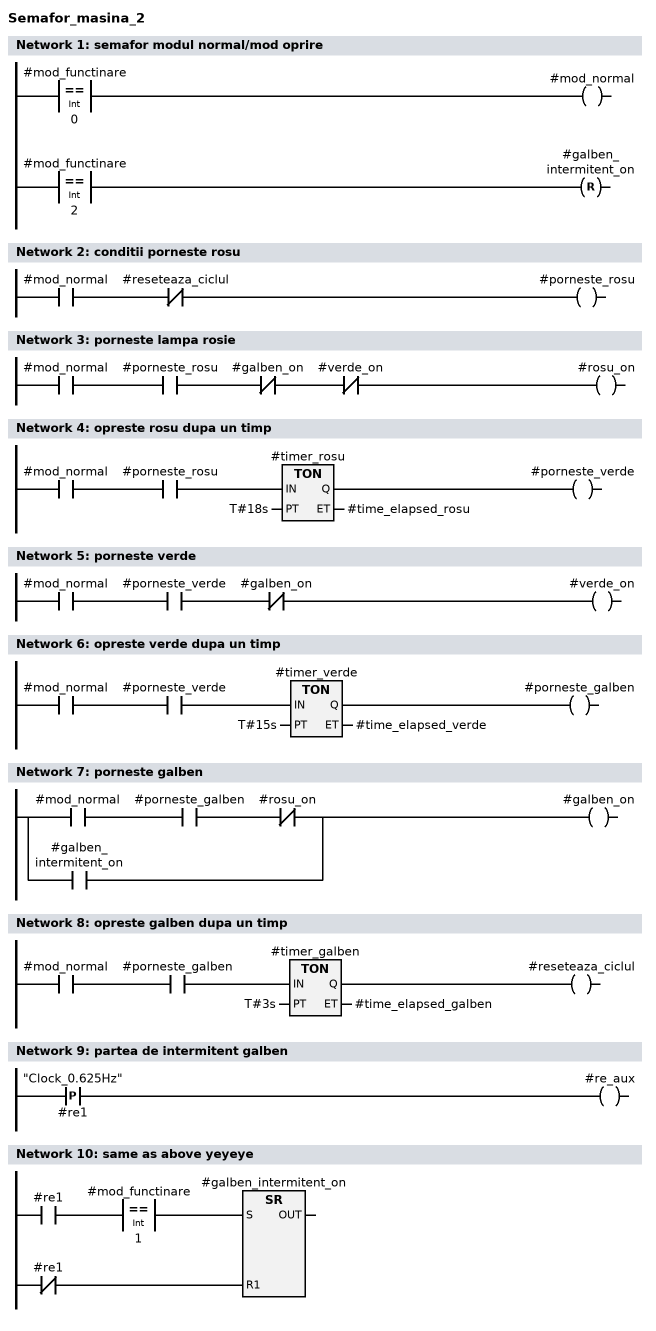
   RUNG wire#powerrail
      { S7_Templates := "SrcType := Int" } EQ_Contact(in1 := #mod_functinare, in2 := 0)
      Coil( #mod_normal )
   END_RUNG
   RUNG wire#powerrail
      { S7_Templates := "SrcType := Int" } EQ_Contact(in1 := #mod_functinare, in2 := 2)
      R_Coil( #galben_intermitent_on )
   END_RUNG
   // the same network as SCL:
   #mod_normal := #mod_functinare = 0;
   IF #mod_functinare = 2 THEN #galben_intermitent_on := FALSE; END_IF;
END_REGION

REGION Network 2: conditii porneste rosu
   RUNG wire#powerrail
      Contact( #mod_normal )
      I_Contact( #reseteaza_ciclul )
      Coil( #porneste_rosu )
   END_RUNG
   // the same network as SCL:
   #porneste_rosu := #mod_normal AND NOT #reseteaza_ciclul;
END_REGION

REGION Network 3: porneste lampa rosie
   RUNG wire#powerrail
      Contact( #mod_normal )
      Contact( #porneste_rosu )
      I_Contact( #galben_on )
      I_Contact( #verde_on )
      Coil( #rosu_on )
   END_RUNG
   // the same network as SCL:
   #rosu_on := #mod_normal AND #porneste_rosu AND NOT #galben_on AND NOT #verde_on;
END_REGION

REGION Network 4: opreste rosu dupa un timp
   #timer_rosu(IN := #mod_normal AND #porneste_rosu, PT := T#18s, ET => #time_elapsed_rosu);   // TON
   #porneste_verde := #timer_rosu.Q;
END_REGION

REGION Network 5: porneste verde
   RUNG wire#powerrail
      Contact( #mod_normal )
      Contact( #porneste_verde )
      I_Contact( #galben_on )
      Coil( #verde_on )
   END_RUNG
   // the same network as SCL:
   #verde_on := #mod_normal AND #porneste_verde AND NOT #galben_on;
END_REGION

REGION Network 6: opreste verde dupa un timp
   #timer_verde(IN := #mod_normal AND #porneste_verde, PT := T#15s, ET => #time_elapsed_verde);   // TON
   #porneste_galben := #timer_verde.Q;
END_REGION

REGION Network 7: porneste galben
   RUNG wire#powerrail
      Contact( #mod_normal )
      Contact( #porneste_galben )
      I_Contact( #rosu_on )
      wire#w1
      Coil( #galben_on )
   END_RUNG
   RUNG wire#powerrail
      Contact( #galben_intermitent_on )
   END_RUNG wire#w1
   // the same network as SCL:
   #galben_on := (#mod_normal AND #porneste_galben AND NOT #rosu_on) OR #galben_intermitent_on;
END_REGION

REGION Network 8: opreste galben dupa un timp
   #timer_galben(IN := #mod_normal AND #porneste_galben, PT := T#3s, ET => #time_elapsed_galben);   // TON
   #reseteaza_ciclul := #timer_galben.Q;
END_REGION

REGION Network 9: partea de intermitent galben
   RUNG wire#powerrail
      P_Contact(operand := "Clock_0.625Hz", bit := #re1)
      Coil( #re_aux )
   END_RUNG
   // the same network as SCL:
   #_w1 := "Clock_0.625Hz" AND NOT #re1;   // rising edge of "Clock_0.625Hz"
   #re1 := "Clock_0.625Hz";
   #re_aux := #_w1;
END_REGION

REGION Network 10: same as above yeyeye
   RUNG wire#powerrail
      Contact( #re1 )
      { S7_Templates := "SrcType := Int" } EQ_Contact(in1 := #mod_functinare, in2 := 1)
      S_SR(operand := #galben_intermitent_on, r1 := wire#w1)
   END_RUNG
   RUNG wire#powerrail
      I_Contact( #re1 )
   END_RUNG wire#w1
   // the same network as SCL:
   IF #re1 AND (#mod_functinare = 1) THEN
       #galben_intermitent_on := TRUE;   // SR flip-flop
   END_IF;
   IF NOT #re1 THEN #galben_intermitent_on := FALSE; END_IF;
END_REGION
END_FUNCTION_BLOCK

ORGANIZATION_BLOCK "Main"   // OB1, LAD, ProgramCycle
TITLE = "Main Program Sweep (Cycle)"
{ S7_Optimized_Access := 'TRUE' }
VERSION : 0.1
   VAR_INPUT
      Initial_Call : Bool;   // Initial call of this OB
      Remanence : Bool;   // =True, if remanent data are available
   END_VAR
   VAR_TEMP   // added for the SCL form of the ladder/FBD networks
      _w1 : Bool;
   END_VAR
BEGIN

REGION Network 1: Semafor masini ciclu
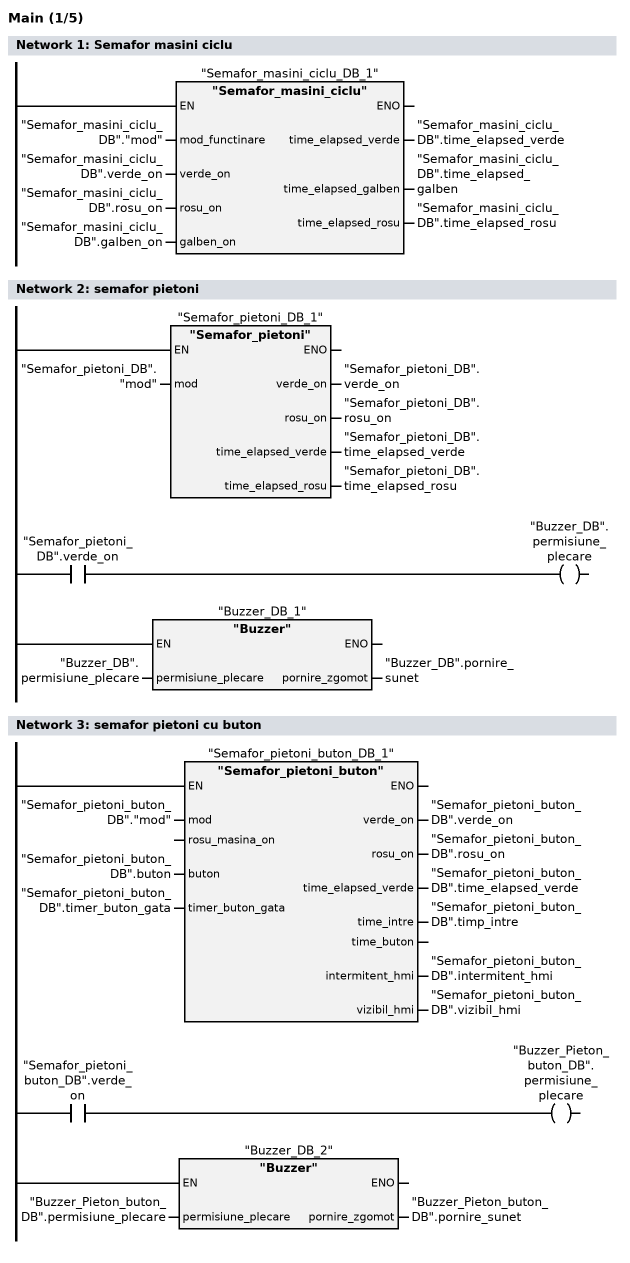
   RUNG wire#powerrail
      "Semafor_masini_ciclu_DB_1"(mod_functinare := "Semafor_masini_ciclu_DB"."mod", verde_on := "Semafor_masini_ciclu_DB".verde_on, rosu_on := "Semafor_masini_ciclu_DB".rosu_on, galben_on := "Semafor_masini_ciclu_DB".galben_on, time_elapsed_verde => "Semafor_masini_ciclu_DB".time_elapsed_verde, time_elapsed_galben => "Semafor_masini_ciclu_DB".time_elapsed_galben, time_elapsed_rosu => "Semafor_masini_ciclu_DB".time_elapsed_rosu)
   END_RUNG
   // the same network as SCL:
   "Semafor_masini_ciclu_DB_1"(mod_functinare := "Semafor_masini_ciclu_DB"."mod",   // "Semafor_masini_ciclu"
                           verde_on := "Semafor_masini_ciclu_DB".verde_on,
                           rosu_on := "Semafor_masini_ciclu_DB".rosu_on,
                           galben_on := "Semafor_masini_ciclu_DB".galben_on,
                           time_elapsed_verde => "Semafor_masini_ciclu_DB".time_elapsed_verde,
                           time_elapsed_galben => "Semafor_masini_ciclu_DB".time_elapsed_galben,
                           time_elapsed_rosu => "Semafor_masini_ciclu_DB".time_elapsed_rosu);
END_REGION

REGION Network 2: semafor pietoni
   RUNG wire#powerrail
      "Semafor_pietoni_DB_1"("mod" := "Semafor_pietoni_DB"."mod", verde_on => "Semafor_pietoni_DB".verde_on, rosu_on => "Semafor_pietoni_DB".rosu_on, time_elapsed_verde => "Semafor_pietoni_DB".time_elapsed_verde, time_elapsed_rosu => "Semafor_pietoni_DB".time_elapsed_rosu)
   END_RUNG
   RUNG wire#powerrail
      Contact( "Semafor_pietoni_DB".verde_on )
      Coil( "Buzzer_DB".permisiune_plecare )
   END_RUNG
   RUNG wire#powerrail
      "Buzzer_DB_1"(permisiune_plecare := "Buzzer_DB".permisiune_plecare, pornire_zgomot => "Buzzer_DB".pornire_sunet)
   END_RUNG
   // the same network as SCL:
   "Semafor_pietoni_DB_1"("mod" := "Semafor_pietoni_DB"."mod",   // "Semafor_pietoni"
                          verde_on => "Semafor_pietoni_DB".verde_on,
                          rosu_on => "Semafor_pietoni_DB".rosu_on,
                          time_elapsed_verde => "Semafor_pietoni_DB".time_elapsed_verde,
                          time_elapsed_rosu => "Semafor_pietoni_DB".time_elapsed_rosu);
   "Buzzer_DB".permisiune_plecare := "Semafor_pietoni_DB".verde_on;
   "Buzzer_DB_1"(permisiune_plecare := "Buzzer_DB".permisiune_plecare,   // "Buzzer"
                 pornire_zgomot => "Buzzer_DB".pornire_sunet);
END_REGION

REGION Network 3: semafor pietoni cu buton
   RUNG wire#powerrail
      "Semafor_pietoni_buton_DB_1"("mod" := "Semafor_pietoni_buton_DB"."mod", rosu_masina_on :=, buton := "Semafor_pietoni_buton_DB".buton, timer_buton_gata := "Semafor_pietoni_buton_DB".timer_buton_gata, verde_on => "Semafor_pietoni_buton_DB".verde_on, rosu_on => "Semafor_pietoni_buton_DB".rosu_on, time_elapsed_verde => "Semafor_pietoni_buton_DB".time_elapsed_verde, time_intre => "Semafor_pietoni_buton_DB".timp_intre, time_buton =>, intermitent_hmi => "Semafor_pietoni_buton_DB".intermitent_hmi, vizibil_hmi => "Semafor_pietoni_buton_DB".vizibil_hmi)
   END_RUNG
   RUNG wire#powerrail
      Contact( "Semafor_pietoni_buton_DB".verde_on )
      Coil( "Buzzer_Pieton_buton_DB".permisiune_plecare )
   END_RUNG
   RUNG wire#powerrail
      "Buzzer_DB_2"(permisiune_plecare := "Buzzer_Pieton_buton_DB".permisiune_plecare, pornire_zgomot => "Buzzer_Pieton_buton_DB".pornire_sunet)
   END_RUNG
   // the same network as SCL:
   "Semafor_pietoni_buton_DB_1"("mod" := "Semafor_pietoni_buton_DB"."mod",   // "Semafor_pietoni_buton"
                           buton := "Semafor_pietoni_buton_DB".buton,
                           timer_buton_gata := "Semafor_pietoni_buton_DB".timer_buton_gata,
                           verde_on => "Semafor_pietoni_buton_DB".verde_on,
                           rosu_on => "Semafor_pietoni_buton_DB".rosu_on,
                           time_elapsed_verde => "Semafor_pietoni_buton_DB".time_elapsed_verde,
                           time_intre => "Semafor_pietoni_buton_DB".timp_intre,
                           intermitent_hmi => "Semafor_pietoni_buton_DB".intermitent_hmi,
                           vizibil_hmi => "Semafor_pietoni_buton_DB".vizibil_hmi);
   "Buzzer_Pieton_buton_DB".permisiune_plecare := "Semafor_pietoni_buton_DB".verde_on;
   "Buzzer_DB_2"(permisiune_plecare := "Buzzer_Pieton_buton_DB".permisiune_plecare,   // "Buzzer"
                 pornire_zgomot => "Buzzer_Pieton_buton_DB".pornire_sunet);
END_REGION

REGION Network 4: semafor masini cu buton
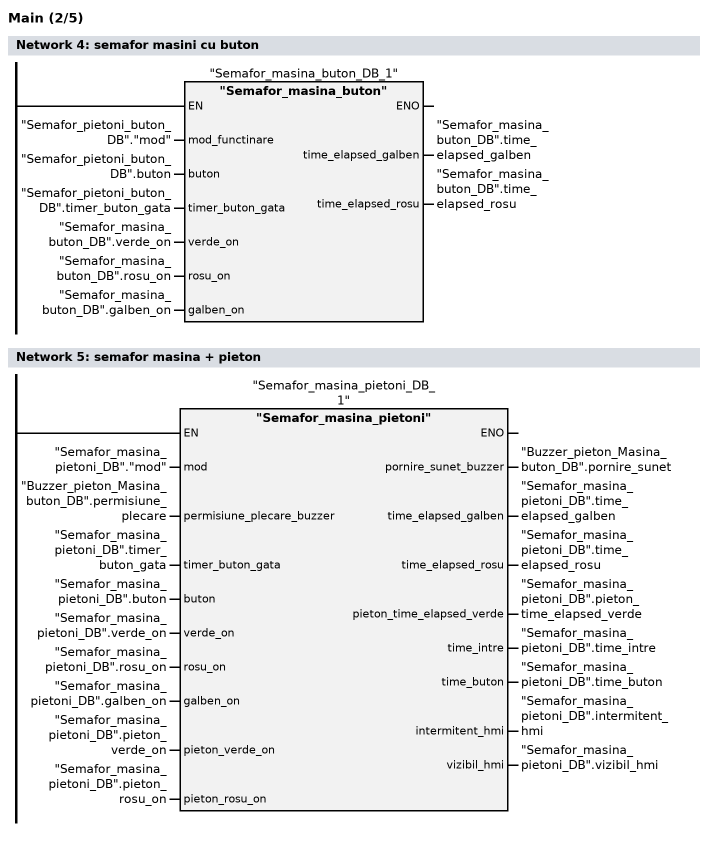
   RUNG wire#powerrail
      "Semafor_masina_buton_DB_1"(mod_functinare := "Semafor_pietoni_buton_DB"."mod", buton := "Semafor_pietoni_buton_DB".buton, timer_buton_gata := "Semafor_pietoni_buton_DB".timer_buton_gata, verde_on := "Semafor_masina_buton_DB".verde_on, rosu_on := "Semafor_masina_buton_DB".rosu_on, galben_on := "Semafor_masina_buton_DB".galben_on, time_elapsed_galben => "Semafor_masina_buton_DB".time_elapsed_galben, time_elapsed_rosu => "Semafor_masina_buton_DB".time_elapsed_rosu)
   END_RUNG
   // the same network as SCL:
   "Semafor_masina_buton_DB_1"(mod_functinare := "Semafor_pietoni_buton_DB"."mod",   // "Semafor_masina_buton"
                           buton := "Semafor_pietoni_buton_DB".buton,
                           timer_buton_gata := "Semafor_pietoni_buton_DB".timer_buton_gata,
                           verde_on := "Semafor_masina_buton_DB".verde_on,
                           rosu_on := "Semafor_masina_buton_DB".rosu_on,
                           galben_on := "Semafor_masina_buton_DB".galben_on,
                           time_elapsed_galben => "Semafor_masina_buton_DB".time_elapsed_galben,
                           time_elapsed_rosu => "Semafor_masina_buton_DB".time_elapsed_rosu);
END_REGION

REGION Network 5: semafor masina + pieton
   RUNG wire#powerrail
      "Semafor_masina_pietoni_DB_1"("mod" := "Semafor_masina_pietoni_DB"."mod", permisiune_plecare_buzzer := "Buzzer_pieton_Masina_buton_DB".permisiune_plecare, timer_buton_gata := "Semafor_masina_pietoni_DB".timer_buton_gata, buton := "Semafor_masina_pietoni_DB".buton, verde_on := "Semafor_masina_pietoni_DB".verde_on, rosu_on := "Semafor_masina_pietoni_DB".rosu_on, galben_on := "Semafor_masina_pietoni_DB".galben_on, pieton_verde_on := "Semafor_masina_pietoni_DB".pieton_verde_on, pieton_rosu_on := "Semafor_masina_pietoni_DB".pieton_rosu_on, pornire_sunet_buzzer => "Buzzer_pieton_Masina_buton_DB".pornire_sunet, time_elapsed_galben => "Semafor_masina_pietoni_DB".time_elapsed_galben, time_elapsed_rosu => "Semafor_masina_pietoni_DB".time_elapsed_rosu, pieton_time_elapsed_verde => "Semafor_masina_pietoni_DB".pieton_time_elapsed_verde, time_intre => "Semafor_masina_pietoni_DB".time_intre, time_buton => "Semafor_masina_pietoni_DB".time_buton, intermitent_hmi => "Semafor_masina_pietoni_DB".intermitent_hmi, vizibil_hmi => "Semafor_masina_pietoni_DB".vizibil_hmi)
   END_RUNG
   // the same network as SCL:
   "Semafor_masina_pietoni_DB_1"("mod" := "Semafor_masina_pietoni_DB"."mod",   // "Semafor_masina_pietoni"
                           permisiune_plecare_buzzer := "Buzzer_pieton_Masina_buton_DB".permisiune_plecare,
                           timer_buton_gata := "Semafor_masina_pietoni_DB".timer_buton_gata,
                           buton := "Semafor_masina_pietoni_DB".buton,
                           verde_on := "Semafor_masina_pietoni_DB".verde_on,
                           rosu_on := "Semafor_masina_pietoni_DB".rosu_on,
                           galben_on := "Semafor_masina_pietoni_DB".galben_on,
                           pieton_verde_on := "Semafor_masina_pietoni_DB".pieton_verde_on,
                           pieton_rosu_on := "Semafor_masina_pietoni_DB".pieton_rosu_on,
                           pornire_sunet_buzzer => "Buzzer_pieton_Masina_buton_DB".pornire_sunet,
                           time_elapsed_galben => "Semafor_masina_pietoni_DB".time_elapsed_galben,
                           time_elapsed_rosu => "Semafor_masina_pietoni_DB".time_elapsed_rosu,
                           pieton_time_elapsed_verde => "Semafor_masina_pietoni_DB".pieton_time_elapsed_verde,
                           time_intre => "Semafor_masina_pietoni_DB".time_intre,
                           time_buton => "Semafor_masina_pietoni_DB".time_buton,
                           intermitent_hmi => "Semafor_masina_pietoni_DB".intermitent_hmi,
                           vizibil_hmi => "Semafor_masina_pietoni_DB".vizibil_hmi);
END_REGION

REGION Network 6: 2 semafoare de masini sincronizate
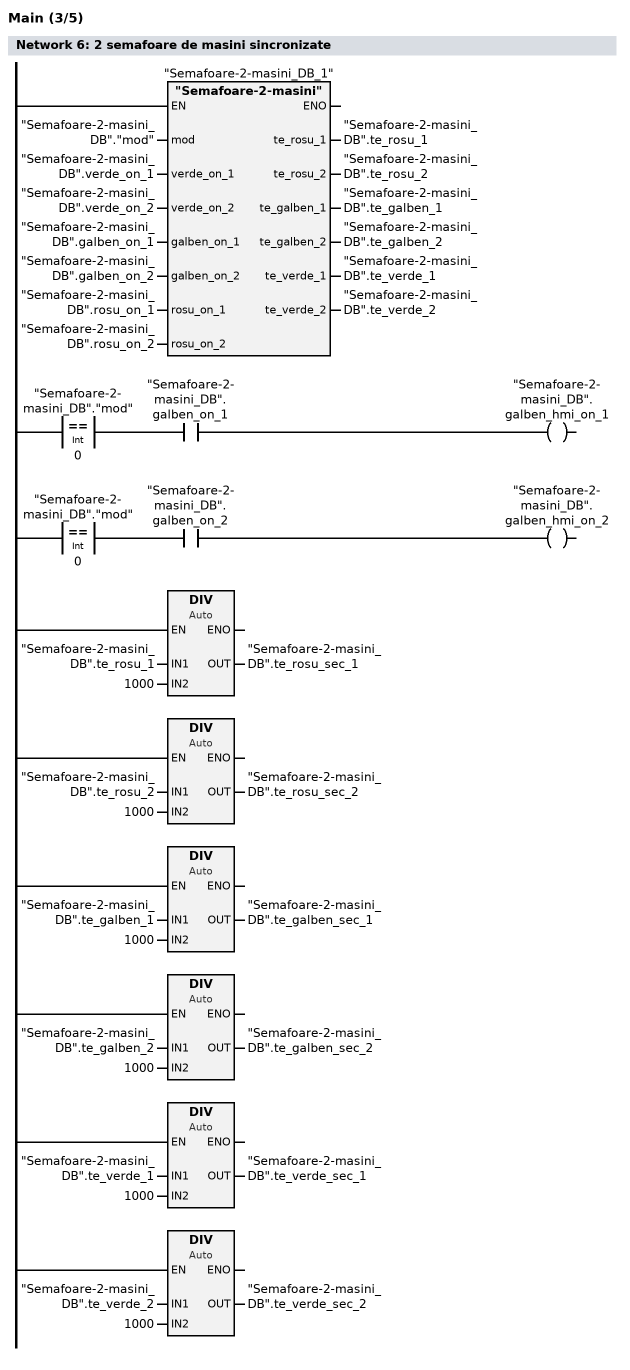
   RUNG wire#powerrail
      "Semafoare-2-masini_DB_1"("mod" := "Semafoare-2-masini_DB"."mod", verde_on_1 := "Semafoare-2-masini_DB".verde_on_1, verde_on_2 := "Semafoare-2-masini_DB".verde_on_2, galben_on_1 := "Semafoare-2-masini_DB".galben_on_1, galben_on_2 := "Semafoare-2-masini_DB".galben_on_2, rosu_on_1 := "Semafoare-2-masini_DB".rosu_on_1, rosu_on_2 := "Semafoare-2-masini_DB".rosu_on_2, te_rosu_1 => "Semafoare-2-masini_DB".te_rosu_1, te_rosu_2 => "Semafoare-2-masini_DB".te_rosu_2, te_galben_1 => "Semafoare-2-masini_DB".te_galben_1, te_galben_2 => "Semafoare-2-masini_DB".te_galben_2, te_verde_1 => "Semafoare-2-masini_DB".te_verde_1, te_verde_2 => "Semafoare-2-masini_DB".te_verde_2)
   END_RUNG
   RUNG wire#powerrail
      { S7_Templates := "SrcType := Int" } EQ_Contact(in1 := "Semafoare-2-masini_DB"."mod", in2 := 0)
      Contact( "Semafoare-2-masini_DB".galben_on_1 )
      Coil( "Semafoare-2-masini_DB".galben_hmi_on_1 )
   END_RUNG
   RUNG wire#powerrail
      { S7_Templates := "SrcType := Int" } EQ_Contact(in1 := "Semafoare-2-masini_DB"."mod", in2 := 0)
      Contact( "Semafoare-2-masini_DB".galben_on_2 )
      Coil( "Semafoare-2-masini_DB".galben_hmi_on_2 )
   END_RUNG
   RUNG wire#powerrail
      Div(in1 := "Semafoare-2-masini_DB".te_rosu_1, in2 := 1000, out => "Semafoare-2-masini_DB".te_rosu_sec_1)
   END_RUNG
   RUNG wire#powerrail
      Div(in1 := "Semafoare-2-masini_DB".te_rosu_2, in2 := 1000, out => "Semafoare-2-masini_DB".te_rosu_sec_2)
   END_RUNG
   RUNG wire#powerrail
      Div(in1 := "Semafoare-2-masini_DB".te_galben_1, in2 := 1000, out => "Semafoare-2-masini_DB".te_galben_sec_1)
   END_RUNG
   RUNG wire#powerrail
      Div(in1 := "Semafoare-2-masini_DB".te_galben_2, in2 := 1000, out => "Semafoare-2-masini_DB".te_galben_sec_2)
   END_RUNG
   RUNG wire#powerrail
      Div(in1 := "Semafoare-2-masini_DB".te_verde_1, in2 := 1000, out => "Semafoare-2-masini_DB".te_verde_sec_1)
   END_RUNG
   RUNG wire#powerrail
      Div(in1 := "Semafoare-2-masini_DB".te_verde_2, in2 := 1000, out => "Semafoare-2-masini_DB".te_verde_sec_2)
   END_RUNG
   // the same network as SCL:
   "Semafoare-2-masini_DB_1"("mod" := "Semafoare-2-masini_DB"."mod",   // "Semafoare-2-masini"
                           verde_on_1 := "Semafoare-2-masini_DB".verde_on_1,
                           verde_on_2 := "Semafoare-2-masini_DB".verde_on_2,
                           galben_on_1 := "Semafoare-2-masini_DB".galben_on_1,
                           galben_on_2 := "Semafoare-2-masini_DB".galben_on_2,
                           rosu_on_1 := "Semafoare-2-masini_DB".rosu_on_1,
                           rosu_on_2 := "Semafoare-2-masini_DB".rosu_on_2,
                           te_rosu_1 => "Semafoare-2-masini_DB".te_rosu_1,
                           te_rosu_2 => "Semafoare-2-masini_DB".te_rosu_2,
                           te_galben_1 => "Semafoare-2-masini_DB".te_galben_1,
                           te_galben_2 => "Semafoare-2-masini_DB".te_galben_2,
                           te_verde_1 => "Semafoare-2-masini_DB".te_verde_1,
                           te_verde_2 => "Semafoare-2-masini_DB".te_verde_2);
   "Semafoare-2-masini_DB".galben_hmi_on_1 := ("Semafoare-2-masini_DB"."mod" = 0) AND "Semafoare-2-masini_DB".galben_on_1;
   "Semafoare-2-masini_DB".galben_hmi_on_2 := ("Semafoare-2-masini_DB"."mod" = 0) AND "Semafoare-2-masini_DB".galben_on_2;
   "Semafoare-2-masini_DB".te_rosu_sec_1 := "Semafoare-2-masini_DB".te_rosu_1 / 1000;
   "Semafoare-2-masini_DB".te_rosu_sec_2 := "Semafoare-2-masini_DB".te_rosu_2 / 1000;
   "Semafoare-2-masini_DB".te_galben_sec_1 := "Semafoare-2-masini_DB".te_galben_1 / 1000;
   "Semafoare-2-masini_DB".te_galben_sec_2 := "Semafoare-2-masini_DB".te_galben_2 / 1000;
   "Semafoare-2-masini_DB".te_verde_sec_1 := "Semafoare-2-masini_DB".te_verde_1 / 1000;
   "Semafoare-2-masini_DB".te_verde_sec_2 := "Semafoare-2-masini_DB".te_verde_2 / 1000;
END_REGION

REGION Network 7: semafor masina-pieton sincronizate
END_REGION

REGION Network 8: intersectie
END_REGION

REGION Network 9: timp in secunde
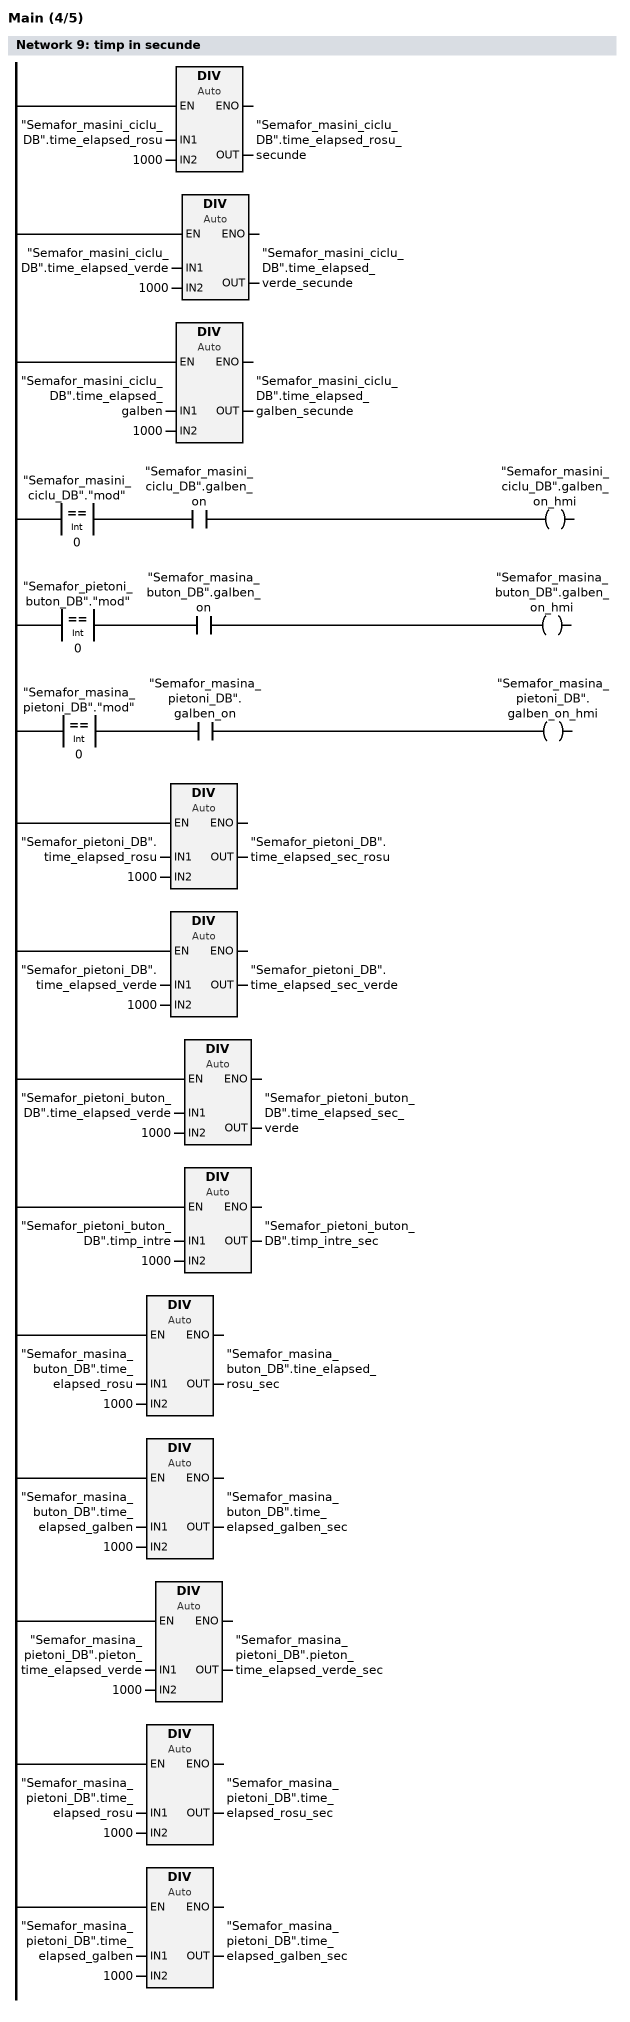
   RUNG wire#powerrail
      Div(in1 := "Semafor_masini_ciclu_DB".time_elapsed_rosu, in2 := 1000, out => "Semafor_masini_ciclu_DB".time_elapsed_rosu_secunde)
   END_RUNG
   RUNG wire#powerrail
      Div(in1 := "Semafor_masini_ciclu_DB".time_elapsed_verde, in2 := 1000, out => "Semafor_masini_ciclu_DB".time_elapsed_verde_secunde)
   END_RUNG
   RUNG wire#powerrail
      Div(in1 := "Semafor_masini_ciclu_DB".time_elapsed_galben, in2 := 1000, out => "Semafor_masini_ciclu_DB".time_elapsed_galben_secunde)
   END_RUNG
   RUNG wire#powerrail
      { S7_Templates := "SrcType := Int" } EQ_Contact(in1 := "Semafor_masini_ciclu_DB"."mod", in2 := 0)
      Contact( "Semafor_masini_ciclu_DB".galben_on )
      Coil( "Semafor_masini_ciclu_DB".galben_on_hmi )
   END_RUNG
   RUNG wire#powerrail
      { S7_Templates := "SrcType := Int" } EQ_Contact(in1 := "Semafor_pietoni_buton_DB"."mod", in2 := 0)
      Contact( "Semafor_masina_buton_DB".galben_on )
      Coil( "Semafor_masina_buton_DB".galben_on_hmi )
   END_RUNG
   RUNG wire#powerrail
      { S7_Templates := "SrcType := Int" } EQ_Contact(in1 := "Semafor_masina_pietoni_DB"."mod", in2 := 0)
      Contact( "Semafor_masina_pietoni_DB".galben_on )
      Coil( "Semafor_masina_pietoni_DB".galben_on_hmi )
   END_RUNG
   RUNG wire#powerrail
      Div(in1 := "Semafor_pietoni_DB".time_elapsed_rosu, in2 := 1000, out => "Semafor_pietoni_DB".time_elapsed_sec_rosu)
   END_RUNG
   RUNG wire#powerrail
      Div(in1 := "Semafor_pietoni_DB".time_elapsed_verde, in2 := 1000, out => "Semafor_pietoni_DB".time_elapsed_sec_verde)
   END_RUNG
   RUNG wire#powerrail
      Div(in1 := "Semafor_pietoni_buton_DB".time_elapsed_verde, in2 := 1000, out => "Semafor_pietoni_buton_DB".time_elapsed_sec_verde)
   END_RUNG
   RUNG wire#powerrail
      Div(in1 := "Semafor_pietoni_buton_DB".timp_intre, in2 := 1000, out => "Semafor_pietoni_buton_DB".timp_intre_sec)
   END_RUNG
   RUNG wire#powerrail
      Div(in1 := "Semafor_masina_buton_DB".time_elapsed_rosu, in2 := 1000, out => "Semafor_masina_buton_DB".tine_elapsed_rosu_sec)
   END_RUNG
   RUNG wire#powerrail
      Div(in1 := "Semafor_masina_buton_DB".time_elapsed_galben, in2 := 1000, out => "Semafor_masina_buton_DB".time_elapsed_galben_sec)
   END_RUNG
   RUNG wire#powerrail
      Div(in1 := "Semafor_masina_pietoni_DB".pieton_time_elapsed_verde, in2 := 1000, out => "Semafor_masina_pietoni_DB".pieton_time_elapsed_verde_sec)
   END_RUNG
   RUNG wire#powerrail
      Div(in1 := "Semafor_masina_pietoni_DB".time_elapsed_rosu, in2 := 1000, out => "Semafor_masina_pietoni_DB".time_elapsed_rosu_sec)
   END_RUNG
   RUNG wire#powerrail
      Div(in1 := "Semafor_masina_pietoni_DB".time_elapsed_galben, in2 := 1000, out => "Semafor_masina_pietoni_DB".time_elapsed_galben_sec)
   END_RUNG
   // the same network as SCL:
   "Semafor_masini_ciclu_DB".time_elapsed_rosu_secunde := "Semafor_masini_ciclu_DB".time_elapsed_rosu / 1000;
   "Semafor_masini_ciclu_DB".time_elapsed_verde_secunde := "Semafor_masini_ciclu_DB".time_elapsed_verde / 1000;
   "Semafor_masini_ciclu_DB".time_elapsed_galben_secunde := "Semafor_masini_ciclu_DB".time_elapsed_galben / 1000;
   "Semafor_masini_ciclu_DB".galben_on_hmi := ("Semafor_masini_ciclu_DB"."mod" = 0) AND "Semafor_masini_ciclu_DB".galben_on;
   "Semafor_masina_buton_DB".galben_on_hmi := ("Semafor_pietoni_buton_DB"."mod" = 0) AND "Semafor_masina_buton_DB".galben_on;
   "Semafor_masina_pietoni_DB".galben_on_hmi := ("Semafor_masina_pietoni_DB"."mod" = 0) AND "Semafor_masina_pietoni_DB".galben_on;
   "Semafor_pietoni_DB".time_elapsed_sec_rosu := "Semafor_pietoni_DB".time_elapsed_rosu / 1000;
   "Semafor_pietoni_DB".time_elapsed_sec_verde := "Semafor_pietoni_DB".time_elapsed_verde / 1000;
   "Semafor_pietoni_buton_DB".time_elapsed_sec_verde := "Semafor_pietoni_buton_DB".time_elapsed_verde / 1000;
   "Semafor_pietoni_buton_DB".timp_intre_sec := "Semafor_pietoni_buton_DB".timp_intre / 1000;
   "Semafor_masina_buton_DB".tine_elapsed_rosu_sec := "Semafor_masina_buton_DB".time_elapsed_rosu / 1000;
   "Semafor_masina_buton_DB".time_elapsed_galben_sec := "Semafor_masina_buton_DB".time_elapsed_galben / 1000;
   "Semafor_masina_pietoni_DB".pieton_time_elapsed_verde_sec := "Semafor_masina_pietoni_DB".pieton_time_elapsed_verde / 1000;
   "Semafor_masina_pietoni_DB".time_elapsed_rosu_sec := "Semafor_masina_pietoni_DB".time_elapsed_rosu / 1000;
   "Semafor_masina_pietoni_DB".time_elapsed_galben_sec := "Semafor_masina_pietoni_DB".time_elapsed_galben / 1000;
END_REGION

REGION Network 10: test pt clock de 0.7hz
   // intentia era ca acesta sa fie folosit in loc de cel de 0.625Hz, insa chiar si acesta e prea rapid pentru HMI, astfel o sa raman la cel initial, acesta o sa ramana doar ca EasterEgg pentru curiosi
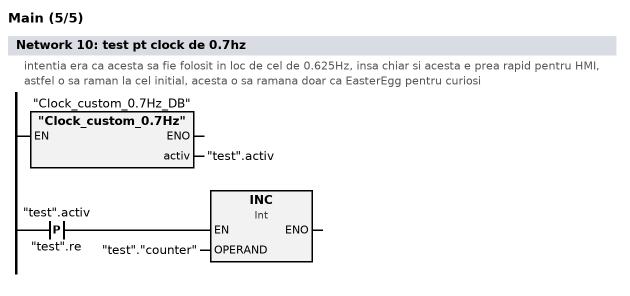
   RUNG wire#powerrail
      "Clock_custom_0.7Hz_DB"(activ => "test".activ)
   END_RUNG
   RUNG wire#powerrail
      P_Contact(operand := "test".activ, bit := "test".re)
      { S7_Templates := "DestType := Int" } Inc( "test"."counter" )
   END_RUNG
   // the same network as SCL:
   "Clock_custom_0.7Hz_DB"(activ => "test".activ);   // "Clock_custom_0.7Hz"
   #_w1 := "test".activ AND NOT "test".re;   // rising edge of "test".activ
   "test".re := "test".activ;
   IF #_w1 THEN "test"."counter" := "test"."counter" + 1; END_IF;
END_REGION
END_ORGANIZATION_BLOCK

(* ===== HMI "HMI_RT_1" =====
system functions are stored by id; their names below are inferred from use
connection "HMI_Connection_1": ETHERNET, SMART_S7_1500_OMS

HMI tags "Default tag table"
   "Semafor_masini_ciclu_DB_rosu_on" : Bool = PLC Semafor_masini_ciclu_DB.rosu_on, 1 s
   "Semafor_masini_ciclu_DB_galben_on" : Bool = PLC Semafor_masini_ciclu_DB.galben_on AT %DB1.DBX0.0, 1 s
   "Semafor_masini_ciclu_DB_verde_on" : Bool = PLC Semafor_masini_ciclu_DB.verde_on AT %DB1.DBX0.0, 1 s
   "Semafor_masini_ciclu_DB_mod" : Int = PLC Semafor_masini_ciclu_DB.mod AT %DB1.DBX0.0, 1 s
   "Semafor_masini_ciclu_DB_time_elapsed_rosu_secunde" : Time = PLC Semafor_masini_ciclu_DB.time_elapsed_rosu_secunde, 1 s
   "Semafor_masini_ciclu_DB_time_elapsed_verde_secunde" : Time = PLC Semafor_masini_ciclu_DB.time_elapsed_verde_secunde, 1 s
   "Semafor_masini_ciclu_DB_time_elapsed_galben_secunde" : Time = PLC Semafor_masini_ciclu_DB.time_elapsed_galben_secunde, 1 s
   "Semafor_masini_ciclu_DB_galben_on_hmi" : Bool = PLC Semafor_masini_ciclu_DB.galben_on_hmi, 1 s
   "Semafor_pietoni_DB_mod" : Int = PLC Semafor_pietoni_DB.mod, 1 s
   "Semafor_pietoni_DB_rosu_on" : Bool = PLC Semafor_pietoni_DB.rosu_on, 1 s
   "Semafor_pietoni_DB_verde_on" : Bool = PLC Semafor_pietoni_DB.verde_on, 1 s
   "Semafor_pietoni_DB_time_elapsed_sec_rosu" : Time = PLC Semafor_pietoni_DB.time_elapsed_sec_rosu, 1 s
   "Semafor_pietoni_DB_time_elapsed_sec_verde" : Time = PLC Semafor_pietoni_DB.time_elapsed_sec_verde, 1 s
   "Semafor_pietoni_buton_mod" : Int = PLC Semafor_pietoni_buton_DB.mod, 1 s
   "Semafor_pietoni_buton_DB_rosu_on" : Bool = PLC Semafor_pietoni_buton_DB.rosu_on, 1 s
   "Semafor_pietoni_buton_DB_verde_on" : Bool = PLC Semafor_pietoni_buton_DB.verde_on, 1 s
   "Semafor_pietoni_buton_DB_time_elapsed_sec_verde" : Time = PLC Semafor_pietoni_buton_DB.time_elapsed_sec_verde, 1 s
   "Semafor_pietoni_buton_DB_buton" : Bool = PLC Semafor_pietoni_buton_DB.buton, 1 s
   "Semafor_pietoni_buton_DB_timp_intre_sec" : Time = PLC Semafor_pietoni_buton_DB.timp_intre_sec, 1 s
   "Semafor_pietoni_buton_DB_intermitent_hmi" : Bool = PLC Semafor_pietoni_buton_DB.intermitent_hmi, 1 s
   "Semafor_pietoni_buton_DB_vizibil_hmi" : Bool = PLC Semafor_pietoni_buton_DB.vizibil_hmi, 1 s
   "Semafor_masina_buton_DB_rosu_on" : Bool = PLC Semafor_masina_buton_DB.rosu_on, 1 s
   "Semafor_masina_buton_DB_galben_on" : Bool = PLC Semafor_masina_buton_DB.galben_on, 1 s
   "Semafor_masina_buton_DB_verde_on" : Bool = PLC Semafor_masina_buton_DB.verde_on, 1 s
   "Semafor_masina_buton_DB_tine_elapsed_rosu_sec" : Time = PLC Semafor_masina_buton_DB.tine_elapsed_rosu_sec, 1 s
   "Semafor_masina_buton_DB_time_elapsed_galben_sec" : Time = PLC Semafor_masina_buton_DB.time_elapsed_galben_sec, 1 s
   "Semafor_masina_buton_DB_galben_on_hmi" : Bool = PLC Semafor_masina_buton_DB.galben_on_hmi, 1 s
   "Semafor_masina_pietoni_DB_mod" : Int = PLC Semafor_masina_pietoni_DB.mod, 1 s
   "Semafor_masina_pietoni_DB_intermitent_hmi" : Bool = PLC Semafor_masina_pietoni_DB.intermitent_hmi, 1 s
   "Semafor_masina_pietoni_DB_buton" : Bool = PLC Semafor_masina_pietoni_DB.buton, 1 s
   "Semafor_masina_pietoni_DB_pieton_verde_on" : Bool = PLC Semafor_masina_pietoni_DB.pieton_verde_on, 1 s
   "Semafor_masina_pietoni_DB_pieton_time_elapsed_verde_sec" : Time = PLC Semafor_masina_pietoni_DB.pieton_time_elapsed_verde_sec, 1 s
   "Semafor_masina_pietoni_DB_pieton_rosu_on" : Bool = PLC Semafor_masina_pietoni_DB.pieton_rosu_on, 1 s
   "Semafor_masina_pietoni_DB_rosu_on" : Bool = PLC Semafor_masina_pietoni_DB.rosu_on, 1 s
   "Semafor_masina_pietoni_DB_galben_on" : Bool = PLC Semafor_masina_pietoni_DB.galben_on, 1 s
   "Semafor_masina_pietoni_DB_verde_on" : Bool = PLC Semafor_masina_pietoni_DB.verde_on, 1 s
   "Semafor_masina_pietoni_DB_time_elapsed_galben_sec" : Time = PLC Semafor_masina_pietoni_DB.time_elapsed_galben_sec, 1 s
   "Semafor_masina_pietoni_DB_time_elapsed_rosu_sec" : Time = PLC Semafor_masina_pietoni_DB.time_elapsed_rosu_sec, 1 s
   "Semafor_masina_pietoni_DB_galben_on_hmi" : Bool = PLC Semafor_masina_pietoni_DB.galben_on_hmi, 1 s
   "Buzzer_DB_pornire_sunet" : Bool = PLC Buzzer_DB.pornire_sunet, 1 s
   "Buzzer_Pieton_buton_DB_pornire_sunet" : Bool = PLC Buzzer_Pieton_buton_DB.pornire_sunet, 1 s
   "Buzzer_pieton_Masina_buton_DB_pornire_sunet" : Bool = PLC Buzzer_pieton_Masina_buton_DB.pornire_sunet, 1 s
   "Semafoare-2-masini_DB_mod" : Int = PLC "Semafoare-2-masini_DB".mod, 1 s
   "Semafoare-2-masini_DB_rosu_on_1" : Bool = PLC "Semafoare-2-masini_DB".rosu_on_1, 1 s
   "Semafoare-2-masini_DB_verde_on_1" : Bool = PLC "Semafoare-2-masini_DB".verde_on_1, 1 s
   "Semafoare-2-masini_DB_galben_hmi_on_1" : Bool = PLC "Semafoare-2-masini_DB".galben_hmi_on_1, 1 s
   "Semafoare-2-masini_DB_galben_hmi_on_2" : Bool = PLC "Semafoare-2-masini_DB".galben_hmi_on_2, 1 s
   "Semafoare-2-masini_DB_verde_on_2" : Bool = PLC "Semafoare-2-masini_DB".verde_on_2, 1 s
   "Semafoare-2-masini_DB_rosu_on_2" : Bool = PLC "Semafoare-2-masini_DB".rosu_on_2, 1 s
   "Semafoare-2-masini_DB_te_rosu_sec_1" : Time = PLC "Semafoare-2-masini_DB".te_rosu_sec_1, 1 s
   "Semafoare-2-masini_DB_te_rosu_sec_2" : Time = PLC "Semafoare-2-masini_DB".te_rosu_sec_2, 1 s
   "Semafoare-2-masini_DB_te_galben_sec_1" : Time = PLC "Semafoare-2-masini_DB".te_galben_sec_1, 1 s
   "Semafoare-2-masini_DB_te_galben_sec_2" : Time = PLC "Semafoare-2-masini_DB".te_galben_sec_2, 1 s
   "Semafoare-2-masini_DB_te_verde_sec_1" : Time = PLC "Semafoare-2-masini_DB".te_verde_sec_1, 1 s
   "Semafoare-2-masini_DB_te_verde_sec_2" : Time = PLC "Semafoare-2-masini_DB".te_verde_sec_2, 1 s
   "Semafoare-2-masini_DB_galben_on_1" : Bool = PLC "Semafoare-2-masini_DB".galben_on_1, 1 s
   "Semafoare-2-masini_DB_galben_on_2" : Bool = PLC "Semafoare-2-masini_DB".galben_on_2, 1 s

text list "Moduri": 0 'Pornit'; 1 'Intermitent'; 2 'Oprit'

Template "Template_1" 800x480
   Button "Exit" at 722,440 size 55x39; TextOff 'Exit'; PictureOff "ExitRuntime_KTP900_Basic_PN_TR"; PictureOn "ExitRuntime_KTP900_Basic_PN_TR"
      on Release: StopRuntime(0)

screen "Semafor_ciclu" 800x480, template "Template_1"
   Circle "Circle_1" at 390,53 size 44x44
      Appearance <- "Semafor_masini_ciclu_DB_rosu_on"
   Circle "Circle_2" at 390,115 size 44x44
      Appearance <- "Semafor_masini_ciclu_DB_galben_on"
   Circle "Circle_3" at 390,178 size 44x44
      Appearance <- "Semafor_masini_ciclu_DB_verde_on"
   Button "Button_1" at 121,86 size 84x32; TextOff 'Pornire'
      on Activate: SetTag("Semafor_masini_ciclu_DB_mod", 0)
      Appearance <- "Semafor_masini_ciclu_DB_mod"
   Button "Button_2" at 121,127 size 84x32; TextOff 'Oprire'
      on Activate: SetTag("Semafor_masini_ciclu_DB_mod", 2)
      Appearance <- "Semafor_masini_ciclu_DB_mod"
   Button "Button_3" at 121,168 size 84x32; TextOff 'Intermitent'
      on Activate: SetTag("Semafor_masini_ciclu_DB_mod", 1)
      Appearance <- "Semafor_masini_ciclu_DB_mod"
   IOField "I/O field_1" at 495,54 size 96x32; FormatPattern 999; Unit s
      ProcessValue <- "Semafor_masini_ciclu_DB_time_elapsed_rosu_secunde"
      Visibility <- "Semafor_masini_ciclu_DB_rosu_on"
   IOField "I/O field_2" at 495,190 size 96x32; FormatPattern 999; Unit s
      ProcessValue <- "Semafor_masini_ciclu_DB_time_elapsed_verde_secunde"
      Visibility <- "Semafor_masini_ciclu_DB_verde_on"
   IOField "I/O field_3" at 495,120 size 96x32; FormatPattern 999; Unit s
      ProcessValue <- "Semafor_masini_ciclu_DB_time_elapsed_galben_secunde"
      Visibility <- "Semafor_masini_ciclu_DB_galben_on_hmi"
   TextField "Text field_1" at 125,451 size 49x20; Text 'Pietoni'
   TextField "Text field_2" at 30,451 size 45x20; Text 'Masini'
   TextField "Text field_3" at 228,451 size 43x20; Text 'Buton'
   TextField "Text field_4" at 313,451 size 77x20; Text 'Intersectie'

screen "Semafor_pieton" 800x480
   Circle "Circle_1" at 383,66 size 57x57
      Appearance <- "Semafor_pietoni_DB_rosu_on"
   Circle "Circle_3" at 383,155 size 57x57
      Appearance <- "Semafor_pietoni_DB_verde_on"
   Button "Button_1" at 121,86 size 84x32; TextOff 'Pornire'
      on Activate: SetTag("Semafor_pietoni_DB_mod", 0)
      Appearance <- "Semafor_pietoni_DB_mod"
   Button "Button_2" at 121,127 size 84x32; TextOff 'Oprire'
      on Activate: SetTag("Semafor_pietoni_DB_mod", 2)
      Appearance <- "Semafor_pietoni_DB_mod"
   IOField "I/O field_1" at 495,76 size 96x32; FormatPattern 999; Unit s
      Visibility <- "Semafor_pietoni_DB_rosu_on"
      ProcessValue <- "Semafor_pietoni_DB_time_elapsed_sec_rosu"
   IOField "I/O field_2" at 495,168 size 96x32; FormatPattern 999; Unit s
      Visibility <- "Semafor_pietoni_DB_verde_on"
      ProcessValue <- "Semafor_pietoni_DB_time_elapsed_sec_verde"
   Rectangle "Rectangle_3" at 274,54 size 39x32
      Visibility <- "Buzzer_DB_pornire_sunet"
   TextField "Text field_5" at 269,30 size 49x20; Text 'Buzzer'
      Visibility <- "Buzzer_DB_pornire_sunet"
   TextField "Text field_1" at 125,451 size 49x20; Text 'Pietoni'
   TextField "Text field_2" at 30,451 size 45x20; Text 'Masini'
   TextField "Text field_3" at 228,451 size 43x20; Text 'Buton'
   TextField "Text field_4" at 313,451 size 77x20; Text 'Intersectie'

screen "Semafor_buton" 800x480
   TextField "Text field_1" at 125,451 size 49x20; Text 'Pietoni'
   TextField "Text field_2" at 30,451 size 45x20; Text 'Masini'
   TextField "Text field_3" at 228,451 size 43x20; Text 'Buton'
   TextField "Text field_4" at 313,451 size 77x20; Text 'Intersectie'
   Button "Button_1" at 105,178 size 44x32; TextOff 'Buton'
      on Click: SetBit("Semafor_masina_pietoni_DB_buton")
      Appearance <- "Semafor_masina_pietoni_DB_intermitent_hmi"
   Circle "Circle_1" at 580,53 size 44x44
      Appearance <- "Semafor_masina_pietoni_DB_rosu_on"
   Circle "Circle_2" at 580,115 size 44x44
      Appearance <- "Semafor_masina_pietoni_DB_galben_on"
   Circle "Circle_3" at 580,178 size 44x44
      Appearance <- "Semafor_masina_pietoni_DB_verde_on"
   IOField "I/O field_3" at 691,54 size 96x32; FormatPattern 999; Unit s
      ProcessValue <- "Semafor_masina_pietoni_DB_time_elapsed_rosu_sec"
      Visibility <- "Semafor_masina_pietoni_DB_rosu_on"
   IOField "I/O field_4" at 691,120 size 96x32; FormatPattern 999; Unit s
      Visibility <- "Semafor_masina_pietoni_DB_galben_on_hmi"
      ProcessValue <- "Semafor_masina_pietoni_DB_time_elapsed_galben_sec"
   TextField "Text field_5" at 570,6 size 62x23; Text 'Masina'
   TextField "Text field_6" at 24,10 size 61x23; Text 'Moduri'
   SymbolicIOField "Symbolic I/O field_1" at 25,38 size 101x37; TextOn '1'; TextOff '0'; TextList "Moduri"
      ProcessValue <- "Semafor_masina_pietoni_DB_mod"
   Circle "Circle_4" at 210,56 size 32x32
      Appearance <- "Semafor_masina_pietoni_DB_pieton_rosu_on"
   Circle "Circle_5" at 210,104 size 33x33
      Appearance <- "Semafor_masina_pietoni_DB_pieton_verde_on"
   IOField "I/O field_2" at 268,106 size 55x32; FormatPattern 999; Unit s
      ProcessValue <- "Semafor_masina_pietoni_DB_pieton_time_elapsed_verde_sec"
      Visibility <- "Semafor_masina_pietoni_DB_pieton_verde_on"
   Rectangle "Rectangle_5" at 185,173 size 83x31
      Appearance <- "Semafor_masina_pietoni_DB_mod"
   TextField "Text field_7" at 185,178 size 80x20; Text 'Intermitent'
   TextField "Text field_8" at 196,10 size 58x23; Text 'Pieton'
   Rectangle "Rectangle_6" at 291,24 size 39x32
      Visibility <- "Buzzer_pieton_Masina_buton_DB_pornire_sunet"
   TextField "Text field_9" at 286,0 size 49x20; Text 'Buzzer'
      Visibility <- "Buzzer_pieton_Masina_buton_DB_pornire_sunet"

screen "Semafor_intersectie" 800x480
   TextField "Text field_1" at 125,451 size 49x20; Text 'Pietoni'
   TextField "Text field_2" at 30,451 size 45x20; Text 'Masini'
   TextField "Text field_3" at 228,451 size 43x20; Text 'Buton'
   TextField "Text field_4" at 313,451 size 77x20; Text 'Intersectie'
   Circle "Circle_1" at 390,53 size 44x44
      Appearance <- "Semafoare-2-masini_DB_rosu_on_1"
   Circle "Circle_2" at 390,115 size 44x44
      Appearance <- "Semafoare-2-masini_DB_galben_on_1"
   Circle "Circle_3" at 390,178 size 44x44
      Appearance <- "Semafoare-2-masini_DB_verde_on_1"
   Button "Button_1" at 121,86 size 84x32; TextOff 'Pornire'
      on Activate: SetTag("Semafoare-2-masini_DB_mod", 0)
      Appearance <- "Semafoare-2-masini_DB_mod"
   Button "Button_2" at 121,127 size 84x32; TextOff 'Oprire'
      on Activate: SetTag("Semafoare-2-masini_DB_mod", 2)
      Appearance <- "Semafoare-2-masini_DB_mod"
   Button "Button_3" at 121,168 size 84x32; TextOff 'Intermitent'
      on Activate: SetTag("Semafoare-2-masini_DB_mod", 1)
      Appearance <- "Semafoare-2-masini_DB_mod"
   IOField "I/O field_1" at 495,54 size 49x32; FormatPattern 999; Unit s
      Visibility <- "Semafoare-2-masini_DB_rosu_on_1"
      ProcessValue <- "Semafoare-2-masini_DB_te_rosu_sec_1"
   IOField "I/O field_2" at 495,190 size 51x32; FormatPattern 999; Unit s
      Visibility <- "Semafoare-2-masini_DB_verde_on_1"
      ProcessValue <- "Semafoare-2-masini_DB_te_verde_sec_1"
   IOField "I/O field_3" at 495,120 size 50x32; FormatPattern 999; Unit s
      Visibility <- "Semafoare-2-masini_DB_galben_hmi_on_1"
      ProcessValue <- "Semafoare-2-masini_DB_te_galben_sec_1"
   Circle "Circle_4" at 631,53 size 44x44
      Appearance <- "Semafoare-2-masini_DB_rosu_on_2"
   Circle "Circle_5" at 631,115 size 44x44
      Appearance <- "Semafoare-2-masini_DB_galben_on_2"
   Circle "Circle_6" at 631,178 size 44x44
      Appearance <- "Semafoare-2-masini_DB_verde_on_2"
   IOField "I/O field_4" at 736,54 size 49x32; FormatPattern 999; Unit s
      Visibility <- "Semafoare-2-masini_DB_rosu_on_2"
      ProcessValue <- "Semafoare-2-masini_DB_te_rosu_sec_2"
   IOField "I/O field_5" at 736,190 size 51x32; FormatPattern 999; Unit s
      Visibility <- "Semafoare-2-masini_DB_verde_on_2"
      ProcessValue <- "Semafoare-2-masini_DB_te_verde_sec_2"
   IOField "I/O field_6" at 736,120 size 50x32; FormatPattern 999; Unit s
      Visibility <- "Semafoare-2-masini_DB_galben_hmi_on_2"
      ProcessValue <- "Semafoare-2-masini_DB_te_galben_sec_2"
   TextField "Text field_5" at 377,10 size 71x20; Text 'Semafor 1'
   TextField "Text field_6" at 619,9 size 71x20; Text 'Semafor 2'
*)